(* IEC 61131-3 sources: SmartHomeNew/snapshots/2026-05-25 (part 2) *)

(* ---- GVL_SENSOR_CONSENSUS.gvl ---- *)
VAR_GLOBAL
    // Global sensor consensus authority.
    Sensor_Consensus_Valid : BOOL := FALSE;
    Sensor_Consensus_Quarantine_Active : BOOL := TRUE;
    Sensor_Consensus_Lease_Expired : BOOL := TRUE;

    // Physics-consistency proofs.
    Physics_Invariants_Satisfied : BOOL := FALSE;
    Cross_Sensor_Correlation_Valid : BOOL := FALSE;
    Telemetry_Plausibility_Valid : BOOL := FALSE;

    // Divergence detection.
    Sensor_Drift_Detected : BOOL := FALSE;
    Sensor_Partition_Detected : BOOL := FALSE;
    Sensor_Hallucination_Suspected : BOOL := FALSE;
    Cross_Sensor_Divergence_Detected : BOOL := FALSE;

    // Physical causality consistency.
    Flow_Response_Valid : BOOL := FALSE;
    Pressure_Response_Valid : BOOL := FALSE;
    Airflow_Response_Valid : BOOL := FALSE;
    Current_Signature_Valid : BOOL := FALSE;

    // Consensus temporal authority.
    Sensor_Consensus_Epoch : UDINT := 0;
    Last_Consensus_Update_MS : UDINT := 0;
    Sensor_Consensus_Freshness_Valid : BOOL := FALSE;

    // Oscillation/drift containment.
    Sensor_Oscillation_Detected : BOOL := FALSE;
    Sensor_Stuck_State_Detected : BOOL := FALSE;
    Sensor_Replay_Suspected : BOOL := FALSE;

    // Diagnostics.
    Sensor_Consensus_Last_Error_Code : UDINT := 0;
    Sensor_Consensus_Last_Error_Text : STRING(160) := '';
    Sensor_Consensus_Invalidation_Count : UDINT := 0;
END_VAR

(* ---- GVL_STATE.gvl ---- *)
{attribute 'qualified_only'}
VAR_GLOBAL
    G_Floor_Temps : ARRAY[1..GVL_CONSTANTS.C_MAX_HEATING_CIRCUITS] OF REAL;
    G_Room_Temps : ARRAY[1..GVL_CONSTANTS.C_MAX_ZONES] OF REAL;
    G_Last_Valid_Room_Temps : ARRAY[1..GVL_CONSTANTS.C_MAX_ZONES] OF REAL;
    G_Last_Valid_Floor_Temps : ARRAY[1..GVL_CONSTANTS.C_MAX_HEATING_CIRCUITS] OF REAL;
    G_Temp_Sensor_Fault : ARRAY[1..GVL_CONSTANTS.C_MAX_ZONES] OF BOOL;
    G_Floor_Temp_Sensor_Fault : ARRAY[1..GVL_CONSTANTS.C_MAX_HEATING_CIRCUITS] OF BOOL;
    G_Room_Hum : ARRAY[1..GVL_CONSTANTS.C_MAX_ZONES] OF REAL;
    G_Room_CO2 : ARRAY[1..GVL_CONSTANTS.C_MAX_ZONES] OF REAL;
    G_Motion_Sensors : ARRAY[1..GVL_CONSTANTS.C_MAX_LIGHT_ZONES] OF BOOL;
    G_Door_Sensors : ARRAY[1..GVL_CONSTANTS.C_MAX_DOOR_SENSORS] OF BOOL;
    G_Window_Sensors : ARRAY[1..GVL_CONSTANTS.C_MAX_ZONES] OF BOOL;
    G_Water_Sensors : ARRAY[1..GVL_CONSTANTS.C_MAX_FLOOD_SENSORS] OF BOOL;
    G_Flood_Warning : ARRAY[1..GVL_CONSTANTS.C_MAX_FLOOD_SENSORS] OF BOOL;
    G_Flood_Alarm : ARRAY[1..GVL_CONSTANTS.C_MAX_FLOOD_SENSORS] OF BOOL;
    G_Flood_Warning_Rise : ARRAY[1..GVL_CONSTANTS.C_MAX_FLOOD_SENSORS] OF BOOL;
    G_Flood_Alarm_Rise : ARRAY[1..GVL_CONSTANTS.C_MAX_FLOOD_SENSORS] OF BOOL;
    G_Flood_Alarm_Fall : ARRAY[1..GVL_CONSTANTS.C_MAX_FLOOD_SENSORS] OF BOOL;
    G_Smoke_Sensors : ARRAY[1..GVL_CONSTANTS.C_MAX_SMOKE_SENSORS] OF BOOL;
    G_Methane_Sensors : ARRAY[1..GVL_CONSTANTS.C_MAX_METHANE_SENSORS] OF REAL;
    G_CO_Sensors : ARRAY[1..GVL_CONSTANTS.C_MAX_CO_SENSORS] OF REAL;
    G_Manifold_Pressures : ARRAY[1..GVL_CONSTANTS.C_MAX_MANIFOLDS] OF REAL;
    G_Manifold_Currents : ARRAY[1..GVL_CONSTANTS.C_MAX_MANIFOLDS] OF REAL;
    G_Predictive_Pump_Pressure_Drop : ARRAY[1..GVL_CONSTANTS.C_MAX_MANIFOLDS] OF BOOL;
    G_Predictive_Pump_Current_Rise : ARRAY[1..GVL_CONSTANTS.C_MAX_MANIFOLDS] OF BOOL;
    G_Manifold_T_Supply : ARRAY[1..GVL_CONSTANTS.C_MAX_MANIFOLDS] OF REAL;
    G_Manifold_T_Return : ARRAY[1..GVL_CONSTANTS.C_MAX_MANIFOLDS] OF REAL;
    G_Boiler_Flame : ARRAY[1..GVL_CONSTANTS.C_MAX_BOILERS] OF BOOL;
    G_Boiler_Error : ARRAY[1..GVL_CONSTANTS.C_MAX_BOILERS] OF BOOL;
    G_Boiler_OT_Online : ARRAY[1..GVL_CONSTANTS.C_MAX_BOILERS] OF BOOL;
    G_Boiler_OT_Command_Ack : ARRAY[1..GVL_CONSTANTS.C_MAX_BOILERS] OF BOOL;
    G_Boiler_OT_Command_Timeout : ARRAY[1..GVL_CONSTANTS.C_MAX_BOILERS] OF BOOL;
    G_Boiler_OT_Heartbeat_Timeout : ARRAY[1..GVL_CONSTANTS.C_MAX_BOILERS] OF BOOL;
    G_Boiler_OT_Adapter_Error : ARRAY[1..GVL_CONSTANTS.C_MAX_BOILERS] OF BOOL;
    G_Boiler_OT_Heartbeat_Age_MS : ARRAY[1..GVL_CONSTANTS.C_MAX_BOILERS] OF UDINT;
    G_Boiler_OT_Command_Age_MS : ARRAY[1..GVL_CONSTANTS.C_MAX_BOILERS] OF UDINT;
    G_Boiler_OT_Adapter_State : ARRAY[1..GVL_CONSTANTS.C_MAX_BOILERS] OF E_OpenTherm_Adapter_State;
    G_Boiler_OT_Error_State : ARRAY[1..GVL_CONSTANTS.C_MAX_BOILERS] OF E_OpenTherm_Error;
    G_Boiler_OT_Enable : ARRAY[1..GVL_CONSTANTS.C_MAX_BOILERS] OF BOOL;
    G_Boiler_OT_Setpoint : ARRAY[1..GVL_CONSTANTS.C_MAX_BOILERS] OF REAL;
    G_Heating_Cascade_Available : BOOL;
    G_Heating_Cascade_Degraded : BOOL;
    G_Heating_Cascade_Partial_Capacity : BOOL;
    G_Heating_Cascade_No_Flame : BOOL;
    G_Heating_Cascade_Transport_Degraded : BOOL;
    G_Heating_Cascade_Ignition_Timeout : BOOL;
    G_Heating_Cascade_Active_Boilers : UINT;
    G_Heating_Cascade_Available_Boilers : UINT;
    G_Physical_Switches : ARRAY[1..GVL_CONSTANTS.C_MAX_LIGHT_ZONES] OF BOOL;
    G_Socket_Switches : ARRAY[1..GVL_CONSTANTS.C_MAX_SOCKETS] OF BOOL;
    G_Outdoor_Temp : REAL;
    G_Ambient_Lux : REAL;
    G_Ambient_Lux_Valid : BOOL := FALSE;
    G_Ambient_Lux_Sensor_Fault : BOOL := FALSE;
    G_Supply_Temps : ARRAY[1..GVL_CONSTANTS.C_MAX_SUPPLY_TEMPS] OF REAL;
    G_DHW_Temp : REAL;
    G_DHW_Pressure : REAL;
    G_Zone_Valves : ARRAY[1..GVL_CONSTANTS.C_MAX_HEATING_CIRCUITS] OF BOOL;
    G_Manifold_Pumps : ARRAY[1..GVL_CONSTANTS.C_MAX_MANIFOLDS] OF BOOL;
    G_Manifold_Valves : ARRAY[1..GVL_CONSTANTS.C_MAX_MANIFOLDS] OF REAL;
    G_Manifold_End_Switches : ARRAY[1..GVL_CONSTANTS.C_MAX_MANIFOLDS] OF BOOL;
    G_Supply_Fans : ARRAY[1..GVL_CONSTANTS.C_MAX_SUPPLY_FANS] OF REAL;
    G_Exhaust_Fans : ARRAY[1..GVL_CONSTANTS.C_MAX_EXHAUST_FANS] OF REAL;
    G_Vent_Heater_Power : ARRAY[1..GVL_CONSTANTS.C_MAX_BOILERS] OF REAL;
    G_Lighting_Levels : ARRAY[1..GVL_CONSTANTS.C_MAX_LIGHT_ZONES] OF BYTE;
    G_Blinds_Positions : ARRAY[1..GVL_CONSTANTS.C_MAX_BLINDS] OF BYTE;
    G_Socket_States : ARRAY[1..GVL_CONSTANTS.C_MAX_SOCKETS] OF BOOL;
    G_DHW_Heating_Pump : BOOL;
    G_DHW_Circ_Pump : BOOL;
    G_Backup_Circulation_Pump : BOOL;
    G_Electric_Heater_Enable : BOOL;
    G_Safety_Gas_Alarm : BOOL;
    G_Safety_Leak_Alarm : BOOL;
    G_Safety_Smoke_Alarm : BOOL;
    G_Safety_Emergency_Stop : BOOL;
    G_Safety_Gas_Latched : BOOL;
    G_Safety_Leak_Latched : BOOL;
    G_Safety_Smoke_Latched : BOOL;
    G_Safety_Freeze_Risk : BOOL;
    G_System_Mode : E_System_Operating_Mode := E_System_Operating_Mode.MODE_NORMAL;
    G_System_Mode_Text : STRING(64);
    G_Heating_IO_Fault : BOOL;
    G_Heating_Sensor_Fault : BOOL;
    G_Heating_Subsystem_Degraded : BOOL;
    G_Allocation_Policy_Active : BOOL;
    G_Allocation_Freeze_Bypass_Active : BOOL;
    G_Allocation_DHW_Bypass_Active : BOOL;
    G_Allocation_Budget_Max : REAL;
    G_Allocation_Budget_Used : REAL;
    G_Allocation_Requested : ARRAY[1..GVL_CONSTANTS.C_MAX_MANIFOLDS] OF BOOL;
    G_Allocation_Allowed : ARRAY[1..GVL_CONSTANTS.C_MAX_MANIFOLDS] OF BOOL;
    G_Allocation_Filtered : ARRAY[1..GVL_CONSTANTS.C_MAX_MANIFOLDS] OF BOOL;
    G_Allocation_Block_Reason : ARRAY[1..GVL_CONSTANTS.C_MAX_MANIFOLDS] OF E_Heating_Allocation_Block_Reason;
    G_Allocation_Effective_Priority : ARRAY[1..GVL_CONSTANTS.C_MAX_MANIFOLDS] OF INT;
    G_Policy_Target_Adjustment_Active : BOOL;
    G_Policy_Target_Adjustment_Applied : REAL;
    G_Policy_Priority_Multiplier_Applied : REAL;
    G_Policy_Priority_Bridge_Active : BOOL;
    G_Policy_Priority_Bias_Applied : ARRAY[1..GVL_CONSTANTS.C_MAX_MANIFOLDS] OF REAL;
    G_Policy_Priority_Effective : ARRAY[1..GVL_CONSTANTS.C_MAX_MANIFOLDS] OF INT;
    G_Heating_RootCause : E_Heating_RootCause := E_Heating_RootCause.RC_NONE;
    G_Heating_RootConfidence : REAL;
    G_Heating_Confidence : REAL := 1.0;
    G_Heating_Error_Score : REAL := 0.0;
    G_Heating_Confidence_Reason_Code : INT := 0;
    G_Heating_Confidence_Reason_Text : STRING(128) := 'OK';
    G_DHW_IO_Fault : BOOL;
    G_DHW_Sensor_Fault : BOOL;
    G_DHW_Subsystem_Degraded : BOOL;
    G_Ventilation_IO_Fault : BOOL;
    G_Ventilation_Subsystem_Degraded : BOOL;
    G_Lighting_IO_Fault : BOOL;
    G_Lighting_Subsystem_Degraded : BOOL;
    G_Access_Comm_Fault : BOOL;
    G_Evacuation_Lighting_Active : BOOL;
    G_Evac_Hazard_Zone : ARRAY[1..GVL_CONSTANTS.C_MAX_LIGHT_ZONES] OF BOOL;
    G_Evac_Guidance : ARRAY[1..GVL_CONSTANTS.C_MAX_LIGHT_ZONES] OF INT;
    G_Rule_Actions : ARRAY[1..GVL_CONSTANTS.C_MAX_RULES] OF ST_Rule_Action;
    G_Sim_Lights : ARRAY[1..GVL_CONSTANTS.C_MAX_LIGHT_ZONES] OF BOOL;
    G_Freeze_Hardware_Degraded : BOOL;
    G_Freeze_Hardware_Failed : BOOL;
    G_Water_Zone_Enable : ARRAY[1..GVL_CONSTANTS.C_MAX_WATER_ZONES] OF BOOL;
    G_Water_Zone_Open_FB : ARRAY[1..GVL_CONSTANTS.C_MAX_WATER_ZONES] OF BOOL;
    G_Water_Zone_Close_FB : ARRAY[1..GVL_CONSTANTS.C_MAX_WATER_ZONES] OF BOOL;
    G_Water_Zone_Exercise_Active : ARRAY[1..GVL_CONSTANTS.C_MAX_WATER_ZONES] OF BOOL;
    G_Preheat_Request : BOOL;
    G_Freeze_Request : BOOL;
    G_Target_Temperature : REAL;
END_VAR

(* ---- GVL_SYSTEM_HEALTH.gvl ---- *)
VAR_GLOBAL
    G_First_Fault_Active : BOOL;
    G_First_Fault_Type : INT;
    G_First_Fault_Source : INT;
    G_System_Severity : E_System_Severity;
    G_Root_Cause : E_System_Root_Cause;
    G_Watchdog_Fault : BOOL;
END_VAR

(* ---- GVL_TIME_SERVICE.gvl ---- *)
{attribute 'qualified_only'}
VAR_GLOBAL
    // Published effective time for consumers
    G_Now_MS : UDINT;
    G_Time_Of_Day_MS : UDINT;
    G_Current_TOD : TOD;
    G_Day_Of_Week : INT;
    G_Last_Now_MS : UDINT;
    G_Delta_MS : UDINT;
    G_Wrap_Detected : BOOL;

    // Simulation controls (HMI/runtime configurable)
    G_Sim_Enabled : BOOL;
    G_Sim_Frozen : BOOL;
    G_Sim_Time_Scale : REAL := 1.0;
    G_Sim_Now_MS : UDINT;
    G_Sim_Time_Of_Day_MS : UDINT;
    G_Sim_Day_Of_Week : INT := 1;
END_VAR

(* ---- GVL_TRUST_EPOCH_MONOTONICITY_FABRIC.gvl ---- *)
VAR_GLOBAL
    // Deterministic trust epoch monotonicity governance.
    Trust_Epoch_Monotonicity_Valid : BOOL := FALSE;
    Trust_Epoch_Monotonicity_Granted : BOOL := FALSE;
    Trust_Epoch_Monotonicity_Quarantine_Active : BOOL := TRUE;

    // Monotonic trust continuity proofs.
    Global_Trust_Epoch_Monotonic : BOOL := FALSE;
    Rollback_Resistant_Authority_Valid : BOOL := FALSE;
    Recovery_Epoch_Strictly_Newer : BOOL := FALSE;
    Distributed_Trust_Vector_Coherent : BOOL := FALSE;
    Irreversible_Trust_Progression_Stable : BOOL := FALSE;

    // Distributed temporal trust integrity.
    CrossNode_Trust_Epoch_Aligned : BOOL := FALSE;
    Recovery_Timeline_Dominance_Valid : BOOL := FALSE;
    Federation_Epoch_Progression_Coherent : BOOL := FALSE;
    Trust_Revocation_History_Monotonic : BOOL := FALSE;

    // Temporal trust rollback detectors.
    Temporal_Trust_Rollback_Detected : BOOL := FALSE;
    Replay_Authority_Epoch_Detected : BOOL := FALSE;
    CrossNode_Trust_Vector_Regression : BOOL := FALSE;
    Stale_Federation_Epoch_Rejoin : BOOL := FALSE;
    Recovery_Timeline_Fork_Detected : BOOL := FALSE;
    Revoked_Epoch_Resurrection_Detected : BOOL := FALSE;

    // Monotonicity epochs.
    Trust_Epoch_Monotonicity_Epoch : UDINT := 0;
    Trust_Epoch_Monotonicity_Epoch_Coherent : BOOL := FALSE;

    // Temporal authority.
    Trust_Epoch_Monotonicity_Last_Update_MS : UDINT := 0;
    Trust_Epoch_Monotonicity_Lease_Expired : BOOL := TRUE;

    // Diagnostics.
    Trust_Epoch_Monotonicity_Last_Error_Code : UDINT := 0;
    Trust_Epoch_Monotonicity_Last_Error_Text : STRING(160) := '';
    Trust_Epoch_Monotonicity_Invalidation_Count : UDINT := 0;
END_VAR

(* ---- GVL_WATER_DOMAIN_STATUS.gvl ---- *)
{attribute 'qualified_only'}
VAR_GLOBAL
    // Water domain status. Observational only.

    G_Runtime_Required : BOOL := FALSE;
    G_Runtime_Executed : BOOL := FALSE;
    G_Runtime_Idle_By_Design : BOOL := FALSE;
    G_Recovery_Requested : BOOL := FALSE;
    G_Global_Path_Active : BOOL := FALSE;
    G_Output_35_Active : BOOL := FALSE;
    G_Output_36_Active : BOOL := FALSE;
    G_Any_Zone_Active : BOOL := FALSE;
    G_Last_Update_MS : UDINT := 0;
    G_Status_Code : UINT := 0;
    G_Status_Text : STRING(128) := '';
END_VAR

(* ---- GVL_Water_Isolation_Intent.gvl ---- *)
{attribute 'qualified_only'}
VAR_GLOBAL
    // ==============================================================================
    // Water/Flood isolation intent publication.
    // ==============================================================================
    //
    // Explicit authority augmentation layer.
    //
    // This layer publishes:
    // - selective isolation intent;
    // - per-zone close requests;
    // - fallback-to-global requirements.
    //
    // It does NOT directly own outputs.
    // Final authority remains inside runtime arbitration/safety layers.
    // ==============================================================================

    // Per-zone isolation intent.
    G_Zone_Close_Requested : ARRAY[1..GVL_CONSTANTS.C_MAX_FLOOD_SENSORS] OF BOOL;

    // Valve-group visibility.
    G_Valve_Group_Close_Requested : ARRAY[1..GVL_CONSTANTS.C_MAX_FLOOD_SENSORS] OF BOOL;

    // Conservative fallback visibility.
    G_Global_Isolation_Requested : BOOL;

    // Explainability.
    G_Intent_Valid : BOOL;
    G_Status_Code : UINT;
    G_Status_Text : STRING(128);
END_VAR

(* ---- GVL_WATER_OUTPUT.gvl ---- *)
VAR_GLOBAL
    // Global inlet valves.
    // 35 = общий ввод ХВС, 36 = общий ввод ГВС.
    DO_Water_Valve_35_Open : BOOL := FALSE;
    DO_Water_Valve_35_Close : BOOL := FALSE;
    DO_Water_Valve_36_Open : BOOL := FALSE;
    DO_Water_Valve_36_Close : BOOL := FALSE;

    // Local riser motorized ball valves with end switches.
    // 1 = стояк 1 ХВС, 2 = стояк 1 ГВС,
    // 3 = стояк 2 ХВС, 4 = стояк 2 ГВС,
    // 5 = стояк 3 ХВС, 6 = стояк 3 ГВС.
    DO_Water_Local_Valve_Open : ARRAY[1..6] OF BOOL;
    DO_Water_Local_Valve_Close : ARRAY[1..6] OF BOOL;

    DO_Water_Zone_Enable : ARRAY[1..GVL_CONSTANTS.C_MAX_WATER_ZONES] OF BOOL;
END_VAR

(* ---- GVL_Water_Topology_Config.gvl ---- *)
{attribute 'qualified_only'}
VAR_GLOBAL
    G_Config_Record : ARRAY[1..64] OF ST_Water_Topology_Config_Record;

    G_Active_Config_Version : UDINT;
    G_Config_Loaded : BOOL;
    G_Runtime_Remap_Ready : BOOL;

    G_Any_Invalid_Config : BOOL;
    G_Any_Multi_Valve_Required : BOOL;

    G_Runtime_Valid : BOOL;
    G_Last_Update_MS : UDINT;

    G_Status_Code : UINT;
    G_Status_Text : STRING(128);
END_VAR

(* ---- GVL_Water_Valve_Runtime.gvl ---- *)
{attribute 'qualified_only'}
VAR_GLOBAL
    // ==============================================================================
    // Water/Flood valve governance publication.
    // ==============================================================================
    //
    // Observe-first valve governance and confirmation visibility.
    //
    // This layer publishes:
    // - valve runtime semantics;
    // - authority visibility;
    // - confirmation semantics;
    // - degraded-state visibility.
    //
    // This layer does NOT directly own physical outputs.
    // ==============================================================================

    G_Valve_Runtime_State : ARRAY[1..64] OF ST_Water_Valve_Runtime_State;

    // Aggregated visibility.
    G_Any_Valve_Degraded : BOOL;
    G_Any_Confirmation_Unknown : BOOL;
    G_Any_Unsafe_Reopen_Denied : BOOL;

    // Lifecycle.
    G_Runtime_Valid : BOOL;
    G_Last_Update_MS : UDINT;

    // Explainability.
    G_Status_Code : UINT;
    G_Status_Text : STRING(128);
END_VAR

(* ---- FB_Access_Pulse_Channel.st ---- *)
FUNCTION_BLOCK FB_Access_Pulse_Channel
VAR_INPUT
    VI_Command : BOOL;
    VI_Reset : BOOL;
    VI_Now_MS : UDINT;
    VI_Pulse_MS : UDINT;
END_VAR
VAR_OUTPUT
    VO_Output : BOOL;
    VO_Active : BOOL;
END_VAR
VAR
    L_Prev_Command : BOOL;
    L_Start_MS : UDINT;
    L_Elapsed_MS : UDINT;
END_VAR

IF VI_Reset THEN
    VO_Output := FALSE;
    VO_Active := FALSE;
    L_Prev_Command := VI_Command;
    L_Start_MS := VI_Now_MS;
    RETURN;
END_IF;

IF VI_Command AND NOT L_Prev_Command THEN
    VO_Active := TRUE;
    L_Start_MS := VI_Now_MS;
END_IF;

VO_Output := FALSE;

IF VO_Active THEN
    IF VI_Now_MS >= L_Start_MS THEN
        L_Elapsed_MS := VI_Now_MS - L_Start_MS;
    ELSE
        L_Elapsed_MS := (4294967295 - L_Start_MS) + VI_Now_MS + 1;
    END_IF;

    IF L_Elapsed_MS < VI_Pulse_MS THEN
        VO_Output := TRUE;
    ELSE
        VO_Active := FALSE;
    END_IF;
END_IF;

L_Prev_Command := VI_Command;

END_FUNCTION_BLOCK
// >>> BULK_SYNC_ANCHOR: FB_Access_Pulse_Channel <<<

(* ---- FB_Alarm_Manager.st ---- *)
FUNCTION_BLOCK FB_Alarm_Manager
VAR_INPUT
    VI_System_Time_MS : UDINT; // Системное время (мс)
    VI_IsActivePLC : BOOL; // Флаг: Данный ПЛК является ведущим

    // Входы от подсистем
    VI_Gas_Alarm : BOOL; // Сигнал тревоги: Утечка газа
    VI_Fire_Alarm : BOOL; // Сигнал тревоги: Пожар
    VI_Flood_Alarm : BOOL; // Сигнал тревоги: Протечка воды
    VI_Security_Alarm : BOOL; // Сигнал тревоги: Охранная система
    VI_First_Fault_Active : BOOL; // Активна защёлкнутая первая причина деградации
    VI_First_Fault_Type : INT; // 1=IO,2=Sensor,3=Comm,4=Subsystem
    VI_First_Fault_Source : INT; // 1=Heating,2=DHW,3=Ventilation,4=Lighting,5=Access

    // Сообщения от подсистем (для детализации)
    VI_Security_Msg : STRING(200); // Детальное сообщение от охранной системы

    // Команды с HMI
    VI_Acknowledge_All : BOOL; // Команда: Квитировать все тревоги
    VI_Mute_Siren : BOOL; // Команда: Временное отключение сирены
END_VAR
VAR_IN_OUT
    VI_Boiler_Errors : ARRAY[1..GVL_CONSTANTS.C_MAX_BOILERS] OF BOOL; // Ошибки котлов
END_VAR
VAR_IN_OUT
    VIO_Next_Alarm_ID : UDINT; // Глобальный счетчик ID тревог
END_VAR
VAR_OUTPUT
    VO_Global_Critical : BOOL; // Есть неквитированные критические аварии
    VO_Global_Warning : BOOL;  // Есть неквитированные предупреждения
    VO_Siren_Active : BOOL;    // Требуется включение сирены
    VO_Active_Count : INT;     // Количество активных тревог
    VO_Unacked_Count : INT;    // Количество неквитированных тревог
    VO_Event_Pulse : BOOL;     // Пульс события для History bridge
    VO_Event_Code : UDINT;     // 1201=ack all, 1202=alarm cleared, 1203=alarm created
    VO_Event_Value : REAL;     // Доп. значение события

    VO_Alarm_List : ARRAY[1..GVL_CONSTANTS.C_MAX_ALARMS] OF ST_Alarm_Record; // Список активных тревог для HMI
END_VAR
VAR
    L_i, L_j, L_k : INT;
    L_Target_Slot : INT;
    L_Min_Pri : INT;
    L_Pending_Alarms : ARRAY[1..10] OF ST_Alarm_Record;
    L_Pending_Count : INT := 0;

    // Фронты и антидребезг для детекции новых тревог
    T_Debounce_Gas : FB_System_Timer;
    T_Debounce_Fire : FB_System_Timer;
    T_Debounce_Flood : FB_System_Timer;
    T_Debounce_Security : FB_System_Timer;
    R_Trig_Gas : R_TRIG;
    R_Trig_Fire : R_TRIG;
    R_Trig_Flood : R_TRIG;
    R_Trig_Security : R_TRIG;
    R_Trig_First_Fault : R_TRIG;
    R_Trig_Boiler : ARRAY[1..GVL_CONSTANTS.C_MAX_BOILERS] OF R_TRIG;
    L_First_Fault_Source_Text : STRING(32);
    L_First_Fault_Type_Text : STRING(32);
    L_Event_Pulse_Latched : BOOL;
END_VAR

VO_Event_Pulse := FALSE;
VO_Event_Code := 0;
VO_Event_Value := 0.0;

// 1. Детекция новых тревог (антидребезг + передний фронт)
T_Debounce_Gas(IN := VI_Gas_Alarm, PT := T#100ms, VI_System_Time_MS := VI_System_Time_MS);
T_Debounce_Fire(IN := VI_Fire_Alarm, PT := T#100ms, VI_System_Time_MS := VI_System_Time_MS);
T_Debounce_Flood(IN := VI_Flood_Alarm, PT := T#500ms, VI_System_Time_MS := VI_System_Time_MS);
T_Debounce_Security(IN := VI_Security_Alarm, PT := T#100ms, VI_System_Time_MS := VI_System_Time_MS);

R_Trig_Gas(CLK := T_Debounce_Gas.Q);
R_Trig_Fire(CLK := T_Debounce_Fire.Q);
R_Trig_Flood(CLK := T_Debounce_Flood.Q);
R_Trig_Security(CLK := T_Debounce_Security.Q);
R_Trig_First_Fault(CLK := VI_First_Fault_Active);
FOR L_i := 1 TO GVL_CONSTANTS.C_MAX_BOILERS DO
    R_Trig_Boiler[L_i](CLK := VI_Boiler_Errors[L_i]);
END_FOR;

// 2. Добавление новых тревог в список (Кольцевой буфер)
L_Pending_Count := 0;
L_Event_Pulse_Latched := FALSE;

IF R_Trig_Gas.Q AND L_Pending_Count < 10 THEN
    L_Pending_Count := L_Pending_Count + 1;
    L_Pending_Alarms[L_Pending_Count].Timestamp_MS := VI_System_Time_MS;
    L_Pending_Alarms[L_Pending_Count].Source := 'Gas';
    L_Pending_Alarms[L_Pending_Count].Source_ID := 0;
    L_Pending_Alarms[L_Pending_Count].Message := 'Критическая концентрация газа!';
    L_Pending_Alarms[L_Pending_Count].Severity := E_ALERT_PRIORITY.ALERT_PRIORITY_CRITICAL;
    L_Pending_Alarms[L_Pending_Count].Is_Active := TRUE;
    L_Pending_Alarms[L_Pending_Count].Is_Acknowledged := FALSE;
END_IF;

IF R_Trig_Fire.Q AND L_Pending_Count < 10 THEN
    L_Pending_Count := L_Pending_Count + 1;
    L_Pending_Alarms[L_Pending_Count].Timestamp_MS := VI_System_Time_MS;
    L_Pending_Alarms[L_Pending_Count].Source := 'Fire';
    L_Pending_Alarms[L_Pending_Count].Source_ID := 0;
    L_Pending_Alarms[L_Pending_Count].Message := 'Обнаружено задымление!';
    L_Pending_Alarms[L_Pending_Count].Severity := E_ALERT_PRIORITY.ALERT_PRIORITY_CRITICAL;
    L_Pending_Alarms[L_Pending_Count].Is_Active := TRUE;
    L_Pending_Alarms[L_Pending_Count].Is_Acknowledged := FALSE;
END_IF;

IF R_Trig_Flood.Q AND L_Pending_Count < 10 THEN
    L_Pending_Count := L_Pending_Count + 1;
    L_Pending_Alarms[L_Pending_Count].Timestamp_MS := VI_System_Time_MS;
    L_Pending_Alarms[L_Pending_Count].Source := 'Flood';
    L_Pending_Alarms[L_Pending_Count].Source_ID := 0;
    L_Pending_Alarms[L_Pending_Count].Message := 'Обнаружена протечка воды!';
    L_Pending_Alarms[L_Pending_Count].Severity := E_ALERT_PRIORITY.ALERT_PRIORITY_CRITICAL;
    L_Pending_Alarms[L_Pending_Count].Is_Active := TRUE;
    L_Pending_Alarms[L_Pending_Count].Is_Acknowledged := FALSE;
END_IF;

IF R_Trig_Security.Q AND L_Pending_Count < 10 THEN
    L_Pending_Count := L_Pending_Count + 1;
    L_Pending_Alarms[L_Pending_Count].Timestamp_MS := VI_System_Time_MS;
    L_Pending_Alarms[L_Pending_Count].Source := 'Security';
    L_Pending_Alarms[L_Pending_Count].Source_ID := 0;
    L_Pending_Alarms[L_Pending_Count].Message := VI_Security_Msg;
    L_Pending_Alarms[L_Pending_Count].Severity := E_ALERT_PRIORITY.ALERT_PRIORITY_CRITICAL;
    L_Pending_Alarms[L_Pending_Count].Is_Active := TRUE;
    L_Pending_Alarms[L_Pending_Count].Is_Acknowledged := FALSE;
END_IF;

IF R_Trig_First_Fault.Q AND L_Pending_Count < 10 THEN
    L_Pending_Count := L_Pending_Count + 1;
    L_Pending_Alarms[L_Pending_Count].Timestamp_MS := VI_System_Time_MS;
    L_Pending_Alarms[L_Pending_Count].Source := 'Diagnostics';
    L_Pending_Alarms[L_Pending_Count].Source_ID := TO_BYTE(VI_First_Fault_Source);

    CASE VI_First_Fault_Type OF
        1: L_First_Fault_Type_Text := 'IO';
        2: L_First_Fault_Type_Text := 'Sensor';
        3: L_First_Fault_Type_Text := 'Comm';
        4: L_First_Fault_Type_Text := 'Subsystem';
        ELSE L_First_Fault_Type_Text := 'Unknown';
    END_CASE;

    CASE VI_First_Fault_Source OF
        1: L_First_Fault_Source_Text := 'Heating';
        2: L_First_Fault_Source_Text := 'DHW';
        3: L_First_Fault_Source_Text := 'Ventilation';
        4: L_First_Fault_Source_Text := 'Lighting';
        5: L_First_Fault_Source_Text := 'Access';
        ELSE L_First_Fault_Source_Text := 'Unknown';
    END_CASE;

    L_Pending_Alarms[L_Pending_Count].Message := CONCAT('Diagnostics root cause: ', CONCAT(L_First_Fault_Source_Text, CONCAT(' / ', L_First_Fault_Type_Text)));
    L_Pending_Alarms[L_Pending_Count].Severity := E_ALERT_PRIORITY.ALERT_PRIORITY_HIGH;
    L_Pending_Alarms[L_Pending_Count].Is_Active := TRUE;
    L_Pending_Alarms[L_Pending_Count].Is_Acknowledged := FALSE;
END_IF;

FOR L_j := 1 TO GVL_CONSTANTS.C_MAX_BOILERS DO
    IF R_Trig_Boiler[L_j].Q AND L_Pending_Count < 10 THEN
        L_Pending_Count := L_Pending_Count + 1;
        L_Pending_Alarms[L_Pending_Count].Timestamp_MS := VI_System_Time_MS;
        L_Pending_Alarms[L_Pending_Count].Source := 'Boiler';
        L_Pending_Alarms[L_Pending_Count].Source_ID := TO_BYTE(L_j);
        L_Pending_Alarms[L_Pending_Count].Message := CONCAT('Авария котла №', INT_TO_STRING(L_j));
        L_Pending_Alarms[L_Pending_Count].Severity := E_ALERT_PRIORITY.ALERT_PRIORITY_HIGH;
        L_Pending_Alarms[L_Pending_Count].Is_Active := TRUE;
        L_Pending_Alarms[L_Pending_Count].Is_Acknowledged := FALSE;
    END_IF;
END_FOR;

// Обработка очереди новых тревог с учетом приоритетов
FOR L_i := 1 TO L_Pending_Count DO

    L_Target_Slot := 0;

    // 1. Ищем пустой слот
    FOR L_k := 1 TO GVL_CONSTANTS.C_MAX_ALARMS DO
        IF VO_Alarm_List[L_k].ID = 0 THEN
            L_Target_Slot := L_k;
            EXIT;
        END_IF;
    END_FOR;

    // 2. Ищем квитированную тревогу с наименьшим приоритетом
    IF L_Target_Slot = 0 THEN
        L_Min_Pri := 999;
        FOR L_k := 1 TO GVL_CONSTANTS.C_MAX_ALARMS DO
            IF VO_Alarm_List[L_k].Is_Acknowledged AND TO_INT(VO_Alarm_List[L_k].Severity) < L_Min_Pri THEN
                L_Min_Pri := TO_INT(VO_Alarm_List[L_k].Severity);
                L_Target_Slot := L_k;
            END_IF;
        END_FOR;
    END_IF;

    // 3. Ищем неквитированную тревогу с наименьшим приоритетом (если он ниже добавляемой)
    IF L_Target_Slot = 0 THEN
        L_Min_Pri := 999;
        FOR L_k := 1 TO GVL_CONSTANTS.C_MAX_ALARMS DO
            IF TO_INT(VO_Alarm_List[L_k].Severity) < L_Min_Pri AND TO_INT(VO_Alarm_List[L_k].Severity) < TO_INT(L_Pending_Alarms[L_i].Severity) THEN
                L_Min_Pri := TO_INT(VO_Alarm_List[L_k].Severity);
                L_Target_Slot := L_k;
            END_IF;
        END_FOR;
    END_IF;

    IF L_Target_Slot = 0 THEN
        // Буфер полон критических неквитированных тревог. Не затираем!
        CONTINUE;
    END_IF;

    VO_Alarm_List[L_Target_Slot] := L_Pending_Alarms[L_i];
    VO_Alarm_List[L_Target_Slot].ID := VIO_Next_Alarm_ID;
    VIO_Next_Alarm_ID := VIO_Next_Alarm_ID + 1;
    IF VIO_Next_Alarm_ID = 0 THEN VIO_Next_Alarm_ID := 1; END_IF;
    IF NOT L_Event_Pulse_Latched THEN
        VO_Event_Pulse := TRUE;
        VO_Event_Code := 1203;
        VO_Event_Value := TO_REAL(VO_Alarm_List[L_Target_Slot].Severity);
        L_Event_Pulse_Latched := TRUE;
    END_IF;
END_FOR;

// 3. Обновление статуса существующих тревог (ушли ли они?)
FOR L_i := 1 TO GVL_CONSTANTS.C_MAX_ALARMS DO
    IF VO_Alarm_List[L_i].ID <> 0 THEN
        IF VO_Alarm_List[L_i].Source = 'Gas' THEN VO_Alarm_List[L_i].Is_Active := VI_Gas_Alarm;
        ELSIF VO_Alarm_List[L_i].Source = 'Fire' THEN VO_Alarm_List[L_i].Is_Active := VI_Fire_Alarm;
        ELSIF VO_Alarm_List[L_i].Source = 'Flood' THEN VO_Alarm_List[L_i].Is_Active := VI_Flood_Alarm;
        ELSIF VO_Alarm_List[L_i].Source = 'Security' THEN VO_Alarm_List[L_i].Is_Active := VI_Security_Alarm;
        ELSIF VO_Alarm_List[L_i].Source = 'Diagnostics' THEN VO_Alarm_List[L_i].Is_Active := VI_First_Fault_Active;
        ELSIF VO_Alarm_List[L_i].Source = 'Boiler' THEN
            IF TO_INT(VO_Alarm_List[L_i].Source_ID) >= 1 AND TO_INT(VO_Alarm_List[L_i].Source_ID) <= GVL_CONSTANTS.C_MAX_BOILERS THEN
                VO_Alarm_List[L_i].Is_Active := VI_Boiler_Errors[TO_INT(VO_Alarm_List[L_i].Source_ID)];
            END_IF;
        END_IF;
    END_IF;
END_FOR;

// 4. Квитирование тревог
IF VI_Acknowledge_All THEN
    FOR L_i := 1 TO GVL_CONSTANTS.C_MAX_ALARMS DO
        IF VO_Alarm_List[L_i].ID <> 0 THEN
            VO_Alarm_List[L_i].Is_Acknowledged := TRUE;
        END_IF;
    END_FOR;

    IF NOT L_Event_Pulse_Latched THEN
        VO_Event_Pulse := TRUE;
        VO_Event_Code := 1201;
        VO_Event_Value := TO_REAL(VO_Unacked_Count);
        L_Event_Pulse_Latched := TRUE;
    END_IF;
END_IF;

// 4.5 Автоквитирование некритичных тревог, если они больше не активны
FOR L_i := 1 TO GVL_CONSTANTS.C_MAX_ALARMS DO
    IF VO_Alarm_List[L_i].ID <> 0 AND NOT VO_Alarm_List[L_i].Is_Active AND NOT VO_Alarm_List[L_i].Is_Acknowledged THEN
        IF VO_Alarm_List[L_i].Severity <> E_ALERT_PRIORITY.ALERT_PRIORITY_CRITICAL THEN
            VO_Alarm_List[L_i].Is_Acknowledged := TRUE;
        END_IF;
    END_IF;
END_FOR;

// 5. Очистка списка (удаление неактивных И квитированных тревог)
// В кольцевом буфере мы просто помечаем слот как пустой (ID = 0), без сдвига массива
FOR L_i := 1 TO GVL_CONSTANTS.C_MAX_ALARMS DO
    IF VO_Alarm_List[L_i].ID <> 0 AND NOT VO_Alarm_List[L_i].Is_Active AND VO_Alarm_List[L_i].Is_Acknowledged THEN
        // Удаляем тревогу
        VO_Alarm_List[L_i].ID := 0;
        IF NOT L_Event_Pulse_Latched THEN
            VO_Event_Pulse := TRUE;
            VO_Event_Code := 1202;
            VO_Event_Value := 0.0;
            L_Event_Pulse_Latched := TRUE;
        END_IF;
    END_IF;
END_FOR;

// 6. Подсчет статистики и формирование глобальных флагов
VO_Global_Critical := FALSE;
VO_Global_Warning := FALSE;
VO_Siren_Active := FALSE;
VO_Active_Count := 0;
VO_Unacked_Count := 0;

FOR L_i := 1 TO GVL_CONSTANTS.C_MAX_ALARMS DO
    IF VO_Alarm_List[L_i].ID <> 0 THEN
        IF VO_Alarm_List[L_i].Is_Active THEN
            VO_Active_Count := VO_Active_Count + 1;
        END_IF;

        IF NOT VO_Alarm_List[L_i].Is_Acknowledged THEN
            VO_Unacked_Count := VO_Unacked_Count + 1;

            IF VO_Alarm_List[L_i].Severity = E_ALERT_PRIORITY.ALERT_PRIORITY_CRITICAL THEN
                VO_Global_Critical := TRUE;
                // Сирена работает только для активных неквитированных критических тревог, если не включен Mute
                IF VO_Alarm_List[L_i].Is_Active AND NOT VI_Mute_Siren THEN
                    VO_Siren_Active := TRUE;
                END_IF;
            ELSIF VO_Alarm_List[L_i].Severity = E_ALERT_PRIORITY.ALERT_PRIORITY_HIGH THEN
                VO_Global_Warning := TRUE;
            END_IF;
        END_IF;
    END_IF;
END_FOR;
// >>> BULK_SYNC_ANCHOR: FB_Alarm_Manager <<<
END_FUNCTION_BLOCK

(* ---- FB_Analog_Validator.st ---- *)
FUNCTION_BLOCK FB_Analog_Validator
VAR_INPUT
    VI_Value : REAL;
    VI_Min_Valid : REAL;
    VI_Max_Valid : REAL;
    VI_Fallback_Mode : INT := 0; // 0: Hold last good, 1: Default value
    VI_Default_Value : REAL := 0.0;
END_VAR
VAR_OUTPUT
    VO_Value : REAL;
    VO_Error : BOOL;
END_VAR
VAR
    L_Last_Good_Value : REAL;
    L_First_Valid : BOOL := FALSE;
END_VAR

IF VI_Value >= VI_Min_Valid AND VI_Value <= VI_Max_Valid THEN
    VO_Error := FALSE;
    VO_Value := VI_Value;
    L_Last_Good_Value := VI_Value;
    L_First_Valid := TRUE;
ELSE
    VO_Error := TRUE;
    IF VI_Fallback_Mode = 1 OR NOT L_First_Valid THEN
        VO_Value := VI_Default_Value;
    ELSE
        VO_Value := L_Last_Good_Value;
    END_IF;
END_IF;
// >>> BULK_SYNC_ANCHOR: FB_Analog_Validator <<<
END_FUNCTION_BLOCK

(* ---- FB_BlackBox_Recorder.st ---- *)
FUNCTION_BLOCK FB_BlackBox_Recorder
VAR_INPUT
    VI_Current_Data : ST_BlackBox_Record;
    VI_Freeze       : BOOL;
    VI_Reset        : BOOL;
END_VAR
VAR_OUTPUT
    VO_Frozen       : BOOL;
    VO_Records_Count: INT;
END_VAR
VAR
    L_Write_Index   : INT := 0;
    L_Initialized   : BOOL := FALSE;
END_VAR

IF NOT L_Initialized THEN
    L_Write_Index := GVL_Retain.G_BlackBox_LastIndex;
    IF L_Write_Index < 0 OR L_Write_Index >= GVL_CONSTANTS.C_MAX_BLACKBOX_RECORDS THEN
        L_Write_Index := 0;
        GVL_Retain.G_BlackBox_LastIndex := 0;
    END_IF;
    L_Initialized := TRUE;
END_IF;

IF VI_Reset THEN
    GVL_Retain.G_BlackBox_Frozen := FALSE;
END_IF;

IF VI_Freeze THEN
    GVL_Retain.G_BlackBox_Frozen := TRUE;
END_IF;

VO_Frozen := GVL_Retain.G_BlackBox_Frozen;

IF NOT GVL_Retain.G_BlackBox_Frozen THEN
    GVL_Retain.G_BlackBox_Buffer[L_Write_Index] := VI_Current_Data;
    GVL_Retain.G_BlackBox_LastIndex := L_Write_Index;

    L_Write_Index := L_Write_Index + 1;
    IF L_Write_Index >= GVL_CONSTANTS.C_MAX_BLACKBOX_RECORDS THEN
        L_Write_Index := 0;
    END_IF;
END_IF;

VO_Records_Count := GVL_CONSTANTS.C_MAX_BLACKBOX_RECORDS;
// >>> BULK_SYNC_ANCHOR: FB_BlackBox_Recorder <<<
END_FUNCTION_BLOCK

(* ---- FB_Config_Simulation.st ---- *)
// ==============================================================================
// Config simulation / validation function block
// Service/commissioning validation utility.
// Does NOT own runtime control and does NOT participate in heating phase runtime.
// ==============================================================================
FUNCTION_BLOCK FB_Config_Simulation
VAR_INPUT
    VI_Enable : BOOL;
    VI_Request : BOOL;
    VI_Confirm : BOOL;
END_VAR
VAR_OUTPUT
    VO_Executed : BOOL;
    VO_Result_OK : BOOL;
    VO_Error_Text : STRING(200);
END_VAR
VAR
    L_Error : BOOL;
END_VAR

VO_Executed := FALSE;
VO_Result_OK := GVL_CONFIG_SIMULATION.G_Simulation_Result_OK;
VO_Error_Text := GVL_CONFIG_SIMULATION.G_Simulation_Error_Text;

IF NOT VI_Enable THEN
    RETURN;
END_IF;

IF VI_Request AND VI_Confirm THEN

    L_Error := FALSE;
    VO_Result_OK := TRUE;
    VO_Error_Text := '';

    // Simulate INPUT constraints
    IF (GVL_CONFIG_CONTROL.STG_Reputation_Learning_Rate < 0.0) OR (GVL_CONFIG_CONTROL.STG_Reputation_Learning_Rate > 1.0) THEN
        VO_Result_OK := FALSE;
        VO_Error_Text := 'Invalid learning rate';
        L_Error := TRUE;
    END_IF;

    // Simulate SCENARIO logic
    IF GVL_CONFIG_CONTROL.STG_Night_Start_Hour = GVL_CONFIG_CONTROL.STG_Night_End_Hour THEN
        VO_Result_OK := FALSE;
        VO_Error_Text := 'Night window invalid';
        L_Error := TRUE;
    END_IF;

    // Simulate SAFETY
    IF GVL_CONFIG_CONTROL.STG_Stabilization_Delay_MS < 1000 THEN
        VO_Result_OK := FALSE;
        VO_Error_Text := 'Recovery delay too small';
        L_Error := TRUE;
    END_IF;

    // Simulate FAIL-SAFE policy
    IF NOT (
        GVL_CONFIG_CONTROL.STG_PLC_Inactive_Close_Gas OR
        GVL_CONFIG_CONTROL.STG_PLC_Inactive_Stop_Boiler OR
        GVL_CONFIG_CONTROL.STG_PLC_Inactive_Block_Heating OR
        GVL_CONFIG_CONTROL.STG_PLC_Inactive_Stop_Vent OR
        GVL_CONFIG_CONTROL.STG_PLC_Inactive_Block_Water
    ) THEN
        VO_Result_OK := FALSE;
        VO_Error_Text := 'Fail-safe disabled';
        L_Error := TRUE;
    END_IF;

    GVL_CONFIG_SIMULATION.G_Simulation_Result_OK := NOT L_Error;
    GVL_CONFIG_SIMULATION.G_Simulation_Error_Text := VO_Error_Text;
    GVL_CONFIG_SIMULATION.G_Simulation_Last_Run_MS := GVL_TIME_SERVICE.G_Now_MS;
    VO_Executed := TRUE;

END_IF;

END_FUNCTION_BLOCK
// >>> BULK_SYNC_ANCHOR: FB_Config_Simulation <<<

(* ---- FB_Distributed_Authority_Arbitration.st ---- *)
FUNCTION_BLOCK FB_Distributed_Authority_Arbitration
VAR_INPUT
    VI_Enable : BOOL;
    VI_System_Time_MS : UDINT;
END_VAR
VAR
    L_State : ST_Distributed_Authority_State;
    L_Lease_Expired : BOOL;

    L_Finalized_Runtime_Continuity : BOOL;
END_VAR

IF NOT VI_Enable THEN
    GVL_Distributed_Authority.G_Runtime_Valid := FALSE;
    RETURN;
END_IF;

L_State.Runtime_Valid := TRUE;
L_State.Runtime_System_Time_MS := VI_System_Time_MS;

L_State.Controller_Id :=
    GVL_Distributed_Runtime.G_Local_Node_State.Controller_Id;

L_State.Runtime_Node_Id :=
    GVL_Distributed_Runtime.G_Local_Node_State.Runtime_Node_Id;

L_State.Authority_Domain_Id :=
    GVL_Distributed_Runtime.G_Local_Node_State.Authority_Domain_Id;

L_State.Authority_Election_Active := TRUE;

L_Lease_Expired :=
    (VI_System_Time_MS - GVL_Distributed_Authority.G_Authority_Lease_Start_MS)
    > GVL_Distributed_Authority.G_Authority_Lease_Duration_MS;

L_State.Authority_Lease_Expired := L_Lease_Expired;
L_State.Authority_Lease_Valid := NOT L_Lease_Expired;

L_State.Replication_Consensus_Healthy :=
    GVL_Distributed_Runtime.G_Distributed_Replication_Healthy;

L_State.Replication_Consensus_Stale :=
    NOT GVL_Distributed_Runtime.G_Distributed_Replication_Healthy;

L_Finalized_Runtime_Continuity :=
    GVL_SEMANTIC_PROGRESS.Semantic_Forward_Progress_Valid
    AND GVL_SEMANTIC_PROGRESS.Semantic_Execution_Continuity_OK
    AND NOT GVL_SEMANTIC_PROGRESS.Semantic_Progress_Lease_Expired
    AND NOT GVL_SEMANTIC_PROGRESS.Semantic_Progress_Quarantine_Active
    AND GVL_RUNTIME_SNAPSHOT.Snapshot_Frozen
    AND GVL_RUNTIME_SNAPSHOT.Snapshot_Publication_Allowed
    AND GVL_RUNTIME_SNAPSHOT.Snapshot_Copy_Valid
    AND GVL_RUNTIME_SNAPSHOT.Snapshot_Isolation_Valid
    AND NOT GVL_RUNTIME_SNAPSHOT.Snapshot_Mutation_Detected
    AND GVL_DISTRIBUTED_SNAPSHOT.Distributed_Publication_Reconciled
    AND GVL_DISTRIBUTED_SNAPSHOT.Distributed_Publication_Freeze_Valid
    AND GVL_DISTRIBUTED_SNAPSHOT.Distributed_Snapshot_Consistent
    AND GVL_DISTRIBUTED_COMMIT.Distributed_Commit_Valid
    AND GVL_DISTRIBUTED_COMMIT.Publication_Prepare_Valid
    AND GVL_DISTRIBUTED_COMMIT.Publication_Commit_Confirmed
    AND NOT GVL_DISTRIBUTED_COMMIT.Peer_Commit_Mismatch
    AND NOT GVL_DISTRIBUTED_COMMIT.Commit_Lease_Expired
    AND GVL_OUTPUT_EPOCH.Output_Publication_Valid
    AND GVL_OUTPUT_EPOCH.Output_Runtime_Epoch_Valid
    AND NOT GVL_OUTPUT_EPOCH.Output_Lease_Expired
    AND NOT GVL_OUTPUT_EPOCH.Output_Forced_Safe_Decay
    AND GVL_COMMAND_VERIFY.PreOutput_Barrier_OK
    AND NOT GVL_COMMAND_VERIFY.PreOutput_Block_IO;

L_State.Distributed_Safety_Barrier_OK :=
    GVL_Runtime_Restart_Continuity.G_Runtime_Valid
    AND NOT GVL_Config_Activation.G_Config_Quarantine_Active
    AND NOT GVL_Distributed_Runtime.G_Split_Brain_Suspected
    AND GVL_IO_Binding_Runtime.G_Runtime_Valid
    AND L_Finalized_Runtime_Continuity;

IF NOT L_State.Distributed_Safety_Barrier_OK THEN

    L_State.Split_Brain_Blocked := TRUE;
    L_State.Authority_Observer_Only := TRUE;

    L_State.Status_Code := 3;
    L_State.Status_Text :=
        'Distributed authority blocked by safety barrier';

ELSIF L_State.Replication_Consensus_Healthy
   AND NOT L_Lease_Expired
   AND L_Finalized_Runtime_Continuity THEN

    L_State.Authority_Master_Elected := TRUE;

    L_State.Recovery_Authority_Allowed := TRUE;
    L_State.Rollback_Authority_Allowed := TRUE;
    L_State.Quarantine_Authority_Allowed := TRUE;

    L_State.Status_Code := 1;
    L_State.Status_Text :=
        'Distributed master authority active';

ELSE

    L_State.Authority_Backup_Elected := TRUE;

    L_State.Status_Code := 2;
    L_State.Status_Text :=
        'Distributed backup authority active';

END_IF;

GVL_Distributed_Authority.G_Authority_State := L_State;

GVL_Distributed_Authority.G_Split_Brain_Blocked :=
    L_State.Split_Brain_Blocked;

GVL_Distributed_Authority.G_Distributed_Safety_Barrier_OK :=
    L_State.Distributed_Safety_Barrier_OK;

GVL_Distributed_Authority.G_Runtime_Valid := TRUE;
GVL_Distributed_Authority.G_Last_Update_MS := VI_System_Time_MS;
GVL_Distributed_Authority.G_Status_Code := L_State.Status_Code;
GVL_Distributed_Authority.G_Status_Text := L_State.Status_Text;

END_FUNCTION_BLOCK

(* ---- FB_Distributed_Recovery_Lock_Runtime.st ---- *)
FUNCTION_BLOCK FB_Distributed_Recovery_Lock_Runtime
VAR_INPUT
    VI_Enable : BOOL;
    VI_System_Time_MS : UDINT;
END_VAR
VAR
    L_Lock : ST_Distributed_Recovery_Lock;
    L_Finalized_Runtime_Continuity : BOOL;
END_VAR

IF NOT VI_Enable THEN
    GVL_Distributed_Recovery_Lock.G_Runtime_Valid := FALSE;
    RETURN;
END_IF;

L_Lock := GVL_Distributed_Recovery_Lock.G_Recovery_Lock;

L_Lock.Runtime_System_Time_MS := VI_System_Time_MS;
L_Lock.Lock_Valid := TRUE;

// Finalized runtime continuity proof chain.
L_Finalized_Runtime_Continuity :=
    GVL_SEMANTIC_PROGRESS.Semantic_Forward_Progress_Valid
    AND GVL_SEMANTIC_PROGRESS.Semantic_Execution_Continuity_OK
    AND NOT GVL_SEMANTIC_PROGRESS.Semantic_Progress_Lease_Expired
    AND NOT GVL_SEMANTIC_PROGRESS.Semantic_Progress_Quarantine_Active
    AND GVL_RUNTIME_SNAPSHOT.Snapshot_Frozen
    AND GVL_RUNTIME_SNAPSHOT.Snapshot_Publication_Allowed
    AND GVL_RUNTIME_SNAPSHOT.Snapshot_Copy_Valid
    AND GVL_RUNTIME_SNAPSHOT.Snapshot_Isolation_Valid
    AND NOT GVL_RUNTIME_SNAPSHOT.Snapshot_Mutation_Detected
    AND GVL_DISTRIBUTED_SNAPSHOT.Distributed_Publication_Reconciled
    AND GVL_DISTRIBUTED_SNAPSHOT.Distributed_Publication_Freeze_Valid
    AND GVL_DISTRIBUTED_SNAPSHOT.Distributed_Snapshot_Consistent
    AND GVL_DISTRIBUTED_COMMIT.Distributed_Commit_Valid
    AND GVL_DISTRIBUTED_COMMIT.Publication_Prepare_Valid
    AND GVL_DISTRIBUTED_COMMIT.Publication_Commit_Confirmed
    AND NOT GVL_DISTRIBUTED_COMMIT.Peer_Commit_Mismatch
    AND NOT GVL_DISTRIBUTED_COMMIT.Commit_Lease_Expired
    AND GVL_OUTPUT_EPOCH.Output_Publication_Valid
    AND GVL_OUTPUT_EPOCH.Output_Runtime_Epoch_Valid
    AND NOT GVL_OUTPUT_EPOCH.Output_Lease_Expired
    AND NOT GVL_OUTPUT_EPOCH.Output_Forced_Safe_Decay
    AND GVL_COMMAND_VERIFY.PreOutput_Barrier_OK
    AND NOT GVL_COMMAND_VERIFY.PreOutput_Block_IO;

// Cluster-exclusive recovery execution lock.
IF GVL_Distributed_Runtime.G_Split_Brain_Suspected
   OR GVL_Distributed_Projection_Ownership.G_Any_Ownership_Conflict
   OR GVL_Runtime_Sessions.G_Any_Stale_Session
   OR NOT L_Finalized_Runtime_Continuity THEN

    L_Lock.Lock_Conflict := TRUE;
    L_Lock.Distributed_Execution_Allowed := FALSE;

    GVL_Distributed_Recovery_Lock.G_Recovery_Execution_Blocked := TRUE;
    GVL_Distributed_Recovery_Lock.G_Rollback_Execution_Blocked := TRUE;
    GVL_Distributed_Recovery_Lock.G_Reopen_Execution_Blocked := TRUE;

    L_Lock.Status_Code := 3;
    L_Lock.Status_Text :=
        'Distributed recovery execution locked';

ELSE

    L_Lock.Recovery_Lock_Active := TRUE;
    L_Lock.Distributed_Execution_Allowed := TRUE;

    GVL_Distributed_Recovery_Lock.G_Recovery_Execution_Blocked := FALSE;
    GVL_Distributed_Recovery_Lock.G_Rollback_Execution_Blocked := FALSE;
    GVL_Distributed_Recovery_Lock.G_Reopen_Execution_Blocked := FALSE;

    L_Lock.Status_Code := 0;
    L_Lock.Status_Text :=
        'Distributed recovery lock healthy';

END_IF;

GVL_Distributed_Recovery_Lock.G_Recovery_Lock := L_Lock;

GVL_Distributed_Recovery_Lock.G_Runtime_Valid := TRUE;
GVL_Distributed_Recovery_Lock.G_Last_Update_MS :=
    VI_System_Time_MS;

GVL_Distributed_Recovery_Lock.G_Status_Code :=
    L_Lock.Status_Code;

GVL_Distributed_Recovery_Lock.G_Status_Text :=
    L_Lock.Status_Text;

END_FUNCTION_BLOCK

(* ---- FB_FloorHeating_Controller.st ---- *)
FUNCTION_BLOCK FB_FloorHeating_Controller
VAR_INPUT
    VI_Current_Temp : REAL;
    VI_Config : ST_FloorHeating_Circuit_Config;
    VI_Tariff : ST_Tariff_Config;
    VI_Current_Hour : UINT;
    VI_IsActivePLC : BOOL;
    VI_System_Time_MS : UDINT;
END_VAR
VAR_OUTPUT
    VO_Pump_Run : BOOL;
    VO_Valve_Pos : REAL; // 0..100%
    VO_Valve_Bool : BOOL; // ШИМ выход для термоэлектрического привода
    VO_Effective_Setpoint : REAL;
END_VAR
VAR
    L_Is_Night : BOOL;
    L_PID : FB_PID_Controller;
    L_Last_Time : UDINT;
    L_Cycle_Time_S : REAL;
    L_PWM_Period_MS : UDINT;
    L_PWM_Duty_MS : UDINT;
    L_Current_Phase_MS : UDINT;
    L_PWM_Start_Time : UDINT;
END_VAR

// Вычисление времени цикла
IF L_Last_Time = 0 THEN
    L_Last_Time := VI_System_Time_MS;
    L_Cycle_Time_S := 1.0;
ELSE
    L_Cycle_Time_S := UDINT_TO_REAL((SEL(VI_System_Time_MS >= L_Last_Time, VI_System_Time_MS - L_Last_Time, (4294967295 - L_Last_Time) + VI_System_Time_MS + 1))) / 1000.0;
    L_Last_Time := VI_System_Time_MS;
END_IF;
IF L_Cycle_Time_S <= 0.0 THEN L_Cycle_Time_S := 0.01; END_IF;

// 1. Определение активного тарифа
IF VI_Tariff.Enabled THEN
    IF VI_Tariff.Night_Start_Hour > VI_Tariff.Night_End_Hour THEN
        // Переход через полночь (например, 23:00 - 07:00)
        L_Is_Night := (VI_Current_Hour >= VI_Tariff.Night_Start_Hour) OR (VI_Current_Hour < VI_Tariff.Night_End_Hour);
    ELSE
        // В пределах одного дня
        L_Is_Night := (VI_Current_Hour >= VI_Tariff.Night_Start_Hour) AND (VI_Current_Hour < VI_Tariff.Night_End_Hour);
    END_IF;
ELSE
    L_Is_Night := FALSE;
END_IF;

// 2. Расчет эффективной уставки
VO_Effective_Setpoint := VI_Config.design_temp;
IF L_Is_Night THEN
    VO_Effective_Setpoint := VO_Effective_Setpoint + VI_Tariff.Boost_Delta;
END_IF;

// 3. ПИД-регулирование
L_PID(
    VI_SetPoint := VO_Effective_Setpoint,
    VI_ProcessValue := VI_Current_Temp,
    VI_Kp := VI_Config.pid_kp,
    VI_Tn := 300.0,
    VI_Tv := 0.0,
    VI_Y_Min := 0.0,
    VI_Y_Max := 100.0,
    VI_Cycle_Time_S := L_Cycle_Time_S,
    VO_Output => VO_Valve_Pos
);

// 4. ШИМ-модуляция для термоэлектрического привода
IF VI_Config.pwm_period_s > 0 THEN
    L_PWM_Period_MS := TO_UDINT(VI_Config.pwm_period_s) * 1000;
ELSE
    L_PWM_Period_MS := 600000; // 10 минут
END_IF;

L_Current_Phase_MS := (SEL(VI_System_Time_MS >= L_PWM_Start_Time, VI_System_Time_MS - L_PWM_Start_Time, (4294967295 - L_PWM_Start_Time) + VI_System_Time_MS + 1));
IF L_Current_Phase_MS >= L_PWM_Period_MS THEN
    L_PWM_Start_Time := VI_System_Time_MS - (L_Current_Phase_MS - L_PWM_Period_MS); // Сохраняем остаток для точности
    L_Current_Phase_MS := (SEL(VI_System_Time_MS >= L_PWM_Start_Time, VI_System_Time_MS - L_PWM_Start_Time, (4294967295 - L_PWM_Start_Time) + VI_System_Time_MS + 1));
END_IF;

L_PWM_Duty_MS := TO_UDINT((VO_Valve_Pos / 100.0) * TO_REAL(L_PWM_Period_MS));

IF VI_IsActivePLC THEN
    VO_Pump_Run := (VO_Valve_Pos > 5.0);

    IF VO_Valve_Pos >= 100.0 THEN
        VO_Valve_Bool := TRUE;
    ELSIF VO_Valve_Pos <= 0.0 THEN
        VO_Valve_Bool := FALSE;
    ELSE
        VO_Valve_Bool := (L_Current_Phase_MS <= L_PWM_Duty_MS);
    END_IF;
ELSE
    VO_Pump_Run := FALSE;
    VO_Valve_Bool := FALSE;
END_IF;
END_FUNCTION_BLOCK

(* ---- FB_Gateway_Interface.st ---- *)
FUNCTION_BLOCK FB_Gateway_Interface
VAR_INPUT
    VI_System_Time_MS           : UDINT;
    VI_Local_PLC_Role           : E_PLC_ROLE;
    VI_Incoming_Command         : ST_Gateway_Command;
    VI_Command_Received         : BOOL;
    VI_Outdoor_Temp             : REAL;
    VI_Security_Armed           : BOOL;
    VI_Flood_Alarm_Active       : BOOL;
    VI_Gas_Alarm_Active         : BOOL;
    VI_Fire_Alarm_Active        : BOOL;
    VI_Methane_Concentration    : REAL;
    VI_Active_Scenario          : E_SCENARIO_TYPE;
    VI_Send_2FA_Req             : BOOL;
    VI_2FA_Code                 : STRING(6);
END_VAR

VAR_IN_OUT
    VI_FloorHeating_Temps       : ARRAY[1..GVL_CONSTANTS.C_MAX_HEATING_CIRCUITS] OF REAL;
    VI_Room_Temps               : ARRAY[1..GVL_CONSTANTS.C_MAX_ZONES] OF REAL;
    VI_Zone_Valve_States        : ARRAY[1..GVL_CONSTANTS.C_MAX_HEATING_CIRCUITS] OF BOOL;
    VI_Manifold_Pressures       : ARRAY[1..GVL_CONSTANTS.C_MAX_MANIFOLDS] OF REAL;
    VI_Manifold_Pump_States     : ARRAY[1..GVL_CONSTANTS.C_MAX_MANIFOLDS] OF BOOL;
    VI_Lighting_Base_Levels     : ARRAY[1..GVL_CONSTANTS.C_MAX_LIGHT_ZONES] OF BYTE;
    VI_Socket_States            : ARRAY[1..GVL_CONSTANTS.C_MAX_SOCKETS] OF BOOL;
    VI_Blinds_Positions         : ARRAY[1..GVL_CONSTANTS.C_MAX_BLINDS] OF BYTE;
    VI_Allowed_IPs              : ARRAY[1..GVL_CONSTANTS.C_MAX_ALLOWED_IPS] OF STRING(15);
END_VAR

VAR_OUTPUT
    VO_Modbus_Registers         : ARRAY[0..GVL_CONSTANTS.C_MAX_MODBUS_REGISTERS-1] OF WORD;
    VO_Lighting_Override        : ARRAY[1..GVL_CONSTANTS.C_MAX_LIGHT_ZONES] OF BYTE;
    VO_Blinds_Override          : ARRAY[1..GVL_CONSTANTS.C_MAX_BLINDS] OF BYTE;
    VO_Socket_Override          : ARRAY[1..GVL_CONSTANTS.C_MAX_SOCKETS] OF BOOL;
    VO_Arm_Req                  : BOOL;
    VO_Disarm_Req               : BOOL;
    VO_PIN_Code                 : STRING(4);
    VO_RFID_Tag                 : STRING(20);
    VO_2FA_Code_In              : STRING(6);
    VO_Data_Ready               : BOOL;
    VO_HMI_Status_Message       : STRING(200);
    VO_Telegram_Msg             : STRING(200);
    VO_Send_Telegram            : BOOL;
    VO_Set_Scenario_Req         : BOOL;
    VO_Target_Scenario          : E_SCENARIO_TYPE;
    VO_Set_Temp_Req             : BOOL;
    VO_Target_Zone              : INT;
    VO_Target_Temp              : REAL;
    VO_Set_Vent_Req             : BOOL;
    VO_Target_Vent_Speed        : BYTE;
    VO_Reset_Errors_Req         : BOOL;
    VO_Set_Config_Req           : BOOL;
    VO_Sync_Time_Req            : BOOL;
    VO_New_Time_MS              : UDINT;
END_VAR

VAR
    L_last_update_time          : UDINT;
    L_i                         : INT;
    L_j                         : INT;
    L_idx                       : INT;
    L_tmp_word                  : WORD;
    L_Code_UDINT                : UDINT;
    L_Prev_Fire                 : BOOL;
    L_Prev_Gas                  : BOOL;
    L_Prev_Flood                : BOOL;
    L_Prev_Security             : BOOL;
    L_Deduplicator              : FB_Command_Deduplication;
    L_IP_Allowed                : BOOL;
    L_Process_Command           : ST_Gateway_Command;
    L_Has_Command_To_Process    : BOOL;
END_VAR

VAR RETAIN
    L_Command_Buffer            : ARRAY[1..GVL_CONSTANTS.C_MAX_GATEWAY_COMMANDS] OF ST_Gateway_Command;
    L_Buffer_Head               : INT := 1;
    L_Buffer_Tail               : INT := 1;
    L_Buffer_Count              : INT := 0;
END_VAR

VO_Send_Telegram := FALSE;
IF VI_Fire_Alarm_Active AND NOT L_Prev_Fire THEN
    VO_Telegram_Msg := 'ВНИМАНИЕ! ПОЖАРНАЯ ТРЕВОГА!';
    VO_Send_Telegram := TRUE;
END_IF;
IF VI_Gas_Alarm_Active AND NOT L_Prev_Gas THEN
    VO_Telegram_Msg := 'ВНИМАНИЕ! УТЕЧКА ГАЗА!';
    VO_Send_Telegram := TRUE;
END_IF;
IF VI_Flood_Alarm_Active AND NOT L_Prev_Flood THEN
    VO_Telegram_Msg := 'ВНИМАНИЕ! ПРОТЕЧКА ВОДЫ!';
    VO_Send_Telegram := TRUE;
END_IF;
IF VI_Security_Armed AND NOT L_Prev_Security THEN
    VO_Telegram_Msg := 'ОХРАНА ВКЛЮЧЕНА';
    VO_Send_Telegram := TRUE;
ELSIF NOT VI_Security_Armed AND L_Prev_Security THEN
    VO_Telegram_Msg := 'ОХРАНА ОТКЛЮЧЕНА';
    VO_Send_Telegram := TRUE;
END_IF;

L_Prev_Fire := VI_Fire_Alarm_Active;
L_Prev_Gas := VI_Gas_Alarm_Active;
L_Prev_Flood := VI_Flood_Alarm_Active;
L_Prev_Security := VI_Security_Armed;

IF (VI_System_Time_MS - L_last_update_time) >= GVL_CONSTANTS.C_MS_IN_SECOND THEN
    L_last_update_time := VI_System_Time_MS;
    L_tmp_word := 0;
    IF VI_Local_PLC_Role = E_PLC_ROLE.ROLE_ACTIVE THEN L_tmp_word := L_tmp_word OR 1; END_IF;
    IF VI_Security_Armed THEN L_tmp_word := L_tmp_word OR 2; END_IF;
    IF VI_Flood_Alarm_Active THEN L_tmp_word := L_tmp_word OR 4; END_IF;
    IF VI_Gas_Alarm_Active THEN L_tmp_word := L_tmp_word OR 8; END_IF;
    IF VI_Fire_Alarm_Active THEN L_tmp_word := L_tmp_word OR 16; END_IF;
    VO_Modbus_Registers[0] := L_tmp_word;

    FOR L_i := 1 TO GVL_CONSTANTS.C_MAX_HEATING_CIRCUITS DO
        VO_Modbus_Registers[L_i] := TO_WORD(TO_INT(VI_FloorHeating_Temps[L_i] * REAL#10.0));
    END_FOR;

    FOR L_i := 1 TO GVL_CONSTANTS.C_MAX_ZONES DO
        VO_Modbus_Registers[16 + L_i] := TO_WORD(TO_INT(VI_Room_Temps[L_i] * REAL#10.0));
    END_FOR;

    L_tmp_word := 0;
    FOR L_i := 1 TO GVL_CONSTANTS.C_MAX_HEATING_CIRCUITS DO
        IF VI_Zone_Valve_States[L_i] THEN
            L_tmp_word := L_tmp_word OR SHL(TO_WORD(1), L_i - 1);
        END_IF;
    END_FOR;
    VO_Modbus_Registers[33] := L_tmp_word;

    FOR L_i := 1 TO GVL_CONSTANTS.C_MAX_MANIFOLDS DO
        VO_Modbus_Registers[33 + L_i] := TO_WORD(TO_INT(VI_Manifold_Pressures[L_i] * REAL#100.0));
    END_FOR;

    FOR L_i := 1 TO GVL_CONSTANTS.C_MAX_LIGHT_ZONES DO
        VO_Modbus_Registers[39 + L_i] := TO_WORD(VI_Lighting_Base_Levels[L_i]);
    END_FOR;

    FOR L_i := 1 TO GVL_CONSTANTS.C_MAX_BLINDS DO
        VO_Modbus_Registers[71 + L_i] := TO_WORD(VI_Blinds_Positions[L_i]);
    END_FOR;

    FOR L_i := 0 TO (GVL_CONSTANTS.C_MAX_SOCKETS - 1) / 16 DO
        L_tmp_word := 0;
        FOR L_j := 1 TO 16 DO
            L_idx := (L_i * 16) + L_j;
            IF L_idx <= GVL_CONSTANTS.C_MAX_SOCKETS THEN
                IF VI_Socket_States[L_idx] THEN
                    L_tmp_word := L_tmp_word OR SHL(TO_WORD(1), L_j - 1);
                END_IF;
            END_IF;
        END_FOR;
        VO_Modbus_Registers[92 + L_i] := L_tmp_word;
    END_FOR;

    VO_Modbus_Registers[100] := SEL(VI_Send_2FA_Req, 0, 1);
    IF VI_Send_2FA_Req THEN
        L_Code_UDINT := STRING_TO_UDINT(VI_2FA_Code);
        VO_Modbus_Registers[101] := TO_WORD(L_Code_UDINT AND 16#FFFF);
        VO_Modbus_Registers[102] := TO_WORD(SHR(L_Code_UDINT, 16));
    ELSE
        VO_Modbus_Registers[101] := 0;
        VO_Modbus_Registers[102] := 0;
    END_IF;

    VO_Data_Ready := TRUE;
END_IF;

VO_Arm_Req := FALSE;
VO_Disarm_Req := FALSE;
VO_Set_Scenario_Req := FALSE;
VO_Set_Temp_Req := FALSE;
VO_Set_Vent_Req := FALSE;
VO_Reset_Errors_Req := FALSE;
VO_Set_Config_Req := FALSE;
VO_Sync_Time_Req := FALSE;
L_Has_Command_To_Process := FALSE;

IF VI_Command_Received THEN
    IF VI_Local_PLC_Role = E_PLC_ROLE.ROLE_ACTIVE THEN
        L_Process_Command := VI_Incoming_Command;
        L_Has_Command_To_Process := TRUE;
    ELSE
        IF L_Buffer_Count < GVL_CONSTANTS.C_MAX_GATEWAY_COMMANDS THEN
            L_Command_Buffer[L_Buffer_Head] := VI_Incoming_Command;
            L_Buffer_Head := L_Buffer_Head + 1;
            IF L_Buffer_Head > GVL_CONSTANTS.C_MAX_GATEWAY_COMMANDS THEN L_Buffer_Head := 1; END_IF;
            L_Buffer_Count := L_Buffer_Count + 1;
        END_IF;
    END_IF;
END_IF;

IF NOT L_Has_Command_To_Process AND (VI_Local_PLC_Role = E_PLC_ROLE.ROLE_ACTIVE) AND (L_Buffer_Count > 0) THEN
    L_Process_Command := L_Command_Buffer[L_Buffer_Tail];
    L_Buffer_Tail := L_Buffer_Tail + 1;
    IF L_Buffer_Tail > GVL_CONSTANTS.C_MAX_GATEWAY_COMMANDS THEN L_Buffer_Tail := 1; END_IF;
    L_Buffer_Count := L_Buffer_Count - 1;
    L_Has_Command_To_Process := TRUE;
END_IF;

IF L_Has_Command_To_Process THEN
    L_IP_Allowed := FALSE;
    IF L_Process_Command.source_ip = '' THEN
        L_IP_Allowed := TRUE;
    ELSE
        FOR L_i := 1 TO GVL_CONSTANTS.C_MAX_ALLOWED_IPS DO
            IF VI_Allowed_IPs[L_i] = L_Process_Command.source_ip THEN
                L_IP_Allowed := TRUE;
                EXIT;
            END_IF;
        END_FOR;
    END_IF;

    IF NOT L_IP_Allowed THEN
        VO_HMI_Status_Message := 'Gateway: Ошибка безопасности (Неизвестный IP)';
        RETURN;
    END_IF;

    IF L_Process_Command.crc32 <> DWORD#0 THEN
        VO_HMI_Status_Message := 'Gateway: CRC unsupported in legacy mode';
        RETURN;
    END_IF;

    L_Deduplicator(
        VI_Command_ID := L_Process_Command.command_id,
        VI_Command_Type := L_Process_Command.command_type,
        VI_Command_Value := L_Process_Command.target_value,
        VI_System_Time_MS := VI_System_Time_MS
    );

    IF L_Deduplicator.VO_Is_New_Command THEN
        CASE L_Process_Command.command_type OF
            E_Gateway_Command_Type.CMD_SET_SCENARIO:
                VO_Set_Scenario_Req := TRUE;
                VO_Target_Scenario := L_Process_Command.target_scenario;
                VO_HMI_Status_Message := 'Gateway: Сценарий изменен';
            E_Gateway_Command_Type.CMD_SET_LIGHT:
                IF (L_Process_Command.target_zone >= 1) AND (L_Process_Command.target_zone <= GVL_CONSTANTS.C_MAX_LIGHT_ZONES) THEN
                    VO_Lighting_Override[L_Process_Command.target_zone] := TO_BYTE(L_Process_Command.target_value);
                    VO_HMI_Status_Message := 'Gateway: Команда освещения принята';
                END_IF;
            E_Gateway_Command_Type.CMD_SET_BLINDS:
                IF (L_Process_Command.target_zone >= 1) AND (L_Process_Command.target_zone <= GVL_CONSTANTS.C_MAX_BLINDS) THEN
                    VO_Blinds_Override[L_Process_Command.target_zone] := TO_BYTE(L_Process_Command.target_value);
                    VO_HMI_Status_Message := 'Gateway: Команда штор принята';
                END_IF;
            E_Gateway_Command_Type.CMD_SET_SOCKET:
                IF (L_Process_Command.target_zone >= 1) AND (L_Process_Command.target_zone <= GVL_CONSTANTS.C_MAX_SOCKETS) THEN
                    VO_Socket_Override[L_Process_Command.target_zone] := L_Process_Command.target_on_off;
                    VO_HMI_Status_Message := 'Gateway: Команда розетки принята';
                END_IF;
            E_Gateway_Command_Type.CMD_SET_SECURITY:
                IF L_Process_Command.target_armed THEN VO_Arm_Req := TRUE; ELSE VO_Disarm_Req := TRUE; END_IF;
                VO_PIN_Code := L_Process_Command.target_pin;
                VO_2FA_Code_In := L_Process_Command.target_2fa_code;
                VO_HMI_Status_Message := 'Gateway: Запрос охраны принят';
            E_Gateway_Command_Type.CMD_SET_TEMP:
                IF (L_Process_Command.target_zone >= 1) AND (L_Process_Command.target_zone <= GVL_CONSTANTS.C_MAX_HEATING_CIRCUITS) THEN
                    VO_Set_Temp_Req := TRUE;
                    VO_Target_Zone := L_Process_Command.target_zone;
                    VO_Target_Temp := L_Process_Command.target_value;
                    VO_HMI_Status_Message := 'Gateway: Уставка температуры изменена';
                END_IF;
            E_Gateway_Command_Type.CMD_SET_VENT:
                VO_Set_Vent_Req := TRUE;
                VO_Target_Vent_Speed := TO_BYTE(L_Process_Command.target_value);
                VO_HMI_Status_Message := 'Gateway: Уставка вентиляции изменена';
            E_Gateway_Command_Type.CMD_TELEGRAM_MSG:
                VO_Telegram_Msg := L_Process_Command.telegram_msg;
                VO_Send_Telegram := TRUE;
                VO_HMI_Status_Message := 'Gateway: Сообщение Telegram отправлено';
            E_Gateway_Command_Type.CMD_SYNC_TIME:
                VO_Sync_Time_Req := TRUE;
                VO_New_Time_MS := REAL_TO_UDINT(L_Process_Command.target_value);
                VO_HMI_Status_Message := 'Gateway: Время синхронизировано';
            E_Gateway_Command_Type.CMD_RESET_ERRORS:
                VO_Reset_Errors_Req := TRUE;
                VO_HMI_Status_Message := 'Gateway: Запрос на сброс ошибок принят';
            E_Gateway_Command_Type.CMD_SET_CONFIG:
                VO_Set_Config_Req := TRUE;
                VO_HMI_Status_Message := 'Gateway: Запрос на применение конфигурации принят';
        END_CASE;
    ELSE
        VO_HMI_Status_Message := 'Gateway: duplicate command ignored';
    END_IF;
END_IF;

// >>> BULK_SYNC_ANCHOR: FB_Gateway_Interface <<<
END_FUNCTION_BLOCK

(* ---- FB_Heating_Circuit_Control.st ---- *)
// ==============================================================================
// Heating circuit control helper
//
// Internal refactoring helper for FB_Heating_System_Manager.
// Owns per-circuit sensor validation, temperature source fallback,
// floor-heating controller call, overheat shutdown, and rule action projection.
//
// Temperature source selection is confidence-aware:
// - range invalid still blocks that source;
// - passive input-quality confidence can prefer a healthier fallback;
// - degraded-but-range-valid sources remain operational if no better source exists.
//
// Publishes only canonical runtime projection semantics to
// GVL_Heating_Runtime_Projection. Explainability, predictive observation and
// supervisory ingestion consume that projection downstream.
// ==============================================================================
FUNCTION_BLOCK FB_Heating_Circuit_Control
VAR_INPUT
    VI_System_Time_MS : UDINT;
    VI_Current_Hour : UINT;
    VI_IsActivePLC : BOOL;
    VI_Config : ST_Heating_Config;
    VI_Tariff : ST_Tariff_Config;
    VI_Scenario_Adjust : REAL;
END_VAR

VAR_IN_OUT
    VI_Zone_Configs : ARRAY[1..GVL_CONSTANTS.C_MAX_HEATING_CIRCUITS] OF ST_FloorHeating_Circuit_Config;
    VI_Floor_Temps : ARRAY[1..GVL_CONSTANTS.C_MAX_HEATING_CIRCUITS] OF REAL;
    VI_Room_Temps : ARRAY[1..16] OF REAL;
    VI_Rule_Actions : ARRAY[1..GVL_CONSTANTS.C_MAX_RULES] OF ST_Rule_Action;
END_VAR

VAR_OUTPUT
    VO_Zone_Valves : ARRAY[1..GVL_CONSTANTS.C_MAX_HEATING_CIRCUITS] OF BOOL;
    VO_Heating_Sensor_Fault : BOOL;
END_VAR

VAR
    L_i : INT;
    L_j : INT;
    L_Climate_Zone_ID : INT;
    L_Zone_Config : ST_FloorHeating_Circuit_Config;
    L_Current_Temp : REAL;
    L_Sensor_Error : BOOL;
    L_Floor_Source_Valid : BOOL;
    L_Room_Source_Valid : BOOL;
    L_Floor_Confidence : REAL;
    L_Room_Confidence : REAL;
    L_Min_Source_Confidence : REAL;
    L_Primary_Source_Code : UINT;
    L_Selected_Source_Code : UINT;
    L_Primary_Confidence : REAL;
    L_Fallback_Confidence : REAL;
    L_Selected_Confidence : REAL;
    L_Fallback_Active : BOOL;
    L_Source_Degraded : BOOL;
    L_Reason_Code : UINT;
    L_Reason_Text : STRING(128);
    L_Selected_Source_Text : STRING(64);
    L_Comfort_Target : REAL;
    L_Economy_Target : REAL;
    L_Long_Away_Target : REAL;
    L_Effective_Target : REAL;
    L_Max_Target : REAL;

    L_Prev_Selected_Source_Code : ARRAY[1..GVL_CONSTANTS.C_MAX_HEATING_CIRCUITS] OF UINT;
    L_Prev_Fallback_Active : ARRAY[1..GVL_CONSTANTS.C_MAX_HEATING_CIRCUITS] OF BOOL;
    L_Prev_Source_Loss : ARRAY[1..GVL_CONSTANTS.C_MAX_HEATING_CIRCUITS] OF BOOL;
    L_Source_Loss_Active : BOOL;

    L_Source_Switched_Event : BOOL;
    L_Fallback_Activated_Event : BOOL;
    L_Fallback_Recovered_Event : BOOL;
    L_Source_Loss_Event : BOOL;
    L_Last_Event_Code : UINT;
    L_Last_Event_Text : STRING(128);

    L_Floor_Controllers : ARRAY[1..GVL_CONSTANTS.C_MAX_HEATING_CIRCUITS] OF FB_FloorHeating_Controller;
    L_Overheat_Timer : ARRAY[1..GVL_CONSTANTS.C_MAX_HEATING_CIRCUITS] OF FB_System_Timer;
    fbFloorTempValidator : ARRAY[1..GVL_CONSTANTS.C_MAX_HEATING_CIRCUITS] OF FB_Analog_Validator;
    fbRoomTempValidator : ARRAY[1..16] OF FB_Analog_Validator;
END_VAR

VO_Heating_Sensor_Fault := FALSE;
L_Min_Source_Confidence := GVL_INPUT_VALIDATION_CONFIG.G_Min_Sensor_Confidence;

FOR L_i := 1 TO GVL_CONSTANTS.C_MAX_HEATING_CIRCUITS DO
    fbFloorTempValidator[L_i](
        VI_Value := VI_Floor_Temps[L_i],
        VI_Min_Valid := -40.0,
        VI_Max_Valid := 120.0,
        VI_Fallback_Mode := 0
    );

    L_Climate_Zone_ID := VI_Zone_Configs[L_i].zone;
    IF L_Climate_Zone_ID >= 1 AND L_Climate_Zone_ID <= 16 THEN
        fbRoomTempValidator[L_Climate_Zone_ID](
            VI_Value := VI_Room_Temps[L_Climate_Zone_ID],
            VI_Min_Valid := -40.0,
            VI_Max_Valid := 120.0,
            VI_Fallback_Mode := 0
        );
    END_IF;

    L_Floor_Source_Valid := NOT fbFloorTempValidator[L_i].VO_Error;
    L_Room_Source_Valid :=
        (L_Climate_Zone_ID >= 1) AND
        (L_Climate_Zone_ID <= 16) AND
        (NOT fbRoomTempValidator[L_Climate_Zone_ID].VO_Error);

    L_Floor_Confidence := REAL#1.0;
    IF GVL_INPUT_QUALITY.G_Floor_Temp_Quality[L_i].Quality_Visible THEN
        L_Floor_Confidence := GVL_INPUT_QUALITY.G_Floor_Temp_Quality[L_i].Confidence;
    END_IF;

    L_Room_Confidence := REAL#1.0;
    IF (L_Climate_Zone_ID >= 1) AND (L_Climate_Zone_ID <= 16) THEN
        IF GVL_INPUT_QUALITY.G_Room_Temp_Quality[L_Climate_Zone_ID].Quality_Visible THEN
            L_Room_Confidence := GVL_INPUT_QUALITY.G_Room_Temp_Quality[L_Climate_Zone_ID].Confidence;
        END_IF;
    END_IF;

    IF L_Floor_Confidence < REAL#0.0 THEN
        L_Floor_Confidence := REAL#0.0;
    ELSIF L_Floor_Confidence > REAL#1.0 THEN
        L_Floor_Confidence := REAL#1.0;
    END_IF;

    IF L_Room_Confidence < REAL#0.0 THEN
        L_Room_Confidence := REAL#0.0;
    ELSIF L_Room_Confidence > REAL#1.0 THEN
        L_Room_Confidence := REAL#1.0;
    END_IF;

    // Floor overheat protection remains floor-bound and range-validity based.
    L_Overheat_Timer[L_i](
        IN := L_Floor_Source_Valid AND (fbFloorTempValidator[L_i].VO_Value > VI_Config.Overheat_Threshold),
        PT := T#60s,
        VI_System_Time_MS := VI_System_Time_MS
    );

    L_Current_Temp := REAL#0.0;
    L_Sensor_Error := FALSE;
    L_Selected_Source_Code := 0;
    L_Selected_Source_Text := 'none';
    L_Selected_Confidence := REAL#0.0;
    L_Fallback_Active := FALSE;
    L_Source_Degraded := FALSE;
    L_Reason_Code := 0;
    L_Reason_Text := 'OK';

    IF VI_Zone_Configs[L_i].control_type = 1 OR VI_Zone_Configs[L_i].control_type = 2 THEN
        L_Primary_Source_Code := 1; // room
        L_Primary_Confidence := L_Room_Confidence;
        L_Fallback_Confidence := L_Floor_Confidence;

        // Primary: room air temperature. If room quality is degraded and floor
        // source is healthier, prefer floor fallback without declaring hard fault.
        IF L_Room_Source_Valid AND
           ((L_Room_Confidence >= L_Min_Source_Confidence) OR NOT L_Floor_Source_Valid OR (L_Room_Confidence >= L_Floor_Confidence)) THEN
            L_Current_Temp := fbRoomTempValidator[L_Climate_Zone_ID].VO_Value;
            L_Selected_Source_Code := 1;
            L_Selected_Source_Text := 'room';
            L_Selected_Confidence := L_Room_Confidence;
        ELSIF L_Floor_Source_Valid THEN
            L_Current_Temp := fbFloorTempValidator[L_i].VO_Value;
            L_Selected_Source_Code := 2;
            L_Selected_Source_Text := 'floor';
            L_Selected_Confidence := L_Floor_Confidence;
            L_Fallback_Active := TRUE;
        ELSIF L_Room_Source_Valid THEN
            L_Current_Temp := fbRoomTempValidator[L_Climate_Zone_ID].VO_Value;
            L_Selected_Source_Code := 1;
            L_Selected_Source_Text := 'room';
            L_Selected_Confidence := L_Room_Confidence;
            L_Source_Degraded := TRUE;
            L_Reason_Code := 2;
            L_Reason_Text := 'Room source degraded but retained; floor source unavailable';
        ELSE
            L_Sensor_Error := TRUE;
        END_IF;
    ELSE
        L_Primary_Source_Code := 2; // floor
        L_Primary_Confidence := L_Floor_Confidence;
        L_Fallback_Confidence := L_Room_Confidence;

        // Primary: floor temperature. If floor quality is degraded and room
        // source is healthier, prefer room fallback without declaring hard fault.
        IF L_Floor_Source_Valid AND
           ((L_Floor_Confidence >= L_Min_Source_Confidence) OR NOT L_Room_Source_Valid OR (L_Floor_Confidence >= L_Room_Confidence)) THEN
            L_Current_Temp := fbFloorTempValidator[L_i].VO_Value;
            L_Selected_Source_Code := 2;
            L_Selected_Source_Text := 'floor';
            L_Selected_Confidence := L_Floor_Confidence;
        ELSIF L_Room_Source_Valid THEN
            L_Current_Temp := fbRoomTempValidator[L_Climate_Zone_ID].VO_Value;
            L_Selected_Source_Code := 1;
            L_Selected_Source_Text := 'room';
            L_Selected_Confidence := L_Room_Confidence;
            L_Fallback_Active := TRUE;
        ELSIF L_Floor_Source_Valid THEN
            L_Current_Temp := fbFloorTempValidator[L_i].VO_Value;
            L_Selected_Source_Code := 2;
            L_Selected_Source_Text := 'floor';
            L_Selected_Confidence := L_Floor_Confidence;
            L_Source_Degraded := TRUE;
            L_Reason_Code := 2;
            L_Reason_Text := 'Floor source degraded but retained; room source unavailable';
        ELSE
            L_Sensor_Error := TRUE;
        END_IF;
    END_IF;

    IF L_Fallback_Active THEN
        L_Source_Degraded := TRUE;
        L_Reason_Code := 1;
        IF L_Primary_Source_Code = 1 THEN
            L_Reason_Text := 'Room source degraded or unavailable; floor fallback selected';
        ELSE
            L_Reason_Text := 'Floor source degraded or unavailable; room fallback selected';
        END_IF;
    END_IF;

    IF L_Sensor_Error THEN
        L_Source_Degraded := TRUE;
        L_Reason_Code := 3;
        L_Reason_Text := 'No valid temperature source available';
        VO_Heating_Sensor_Fault := TRUE;
        VO_Zone_Valves[L_i] := FALSE;
    ELSE
        L_Zone_Config := VI_Zone_Configs[L_i];

        IF L_Zone_Config.comfort_temp > REAL#0.0 THEN
            L_Comfort_Target := L_Zone_Config.comfort_temp;
        ELSE
            L_Comfort_Target := L_Zone_Config.design_temp;
        END_IF;

        IF L_Zone_Config.economy_temp > REAL#0.0 THEN
            L_Economy_Target := L_Zone_Config.economy_temp;
        ELSE
            L_Economy_Target := L_Comfort_Target - REAL#3.0;
        END_IF;

        IF L_Zone_Config.long_away_temp > REAL#0.0 THEN
            L_Long_Away_Target := L_Zone_Config.long_away_temp;
        ELSE
            L_Long_Away_Target := GVL_POLICY.G_Away_Long_Economy_Setpoint_C;
        END_IF;

        L_Effective_Target := L_Comfort_Target;

        // Unused rooms may stay in economy even in normal mode.
        IF NOT L_Zone_Config.use_in_normal THEN
            L_Effective_Target := L_Economy_Target;
        END_IF;

        IF GVL_POLICY.G_Away_Active THEN
            CASE GVL_POLICY.G_Away_Level OF
                1:
                    IF L_Zone_Config.use_in_normal THEN
                        L_Effective_Target := L_Comfort_Target + GVL_POLICY.G_Away_Heating_Offset_C;
                    ELSE
                        L_Effective_Target := L_Economy_Target;
                    END_IF;
                2:
                    L_Effective_Target := L_Economy_Target;
                3:
                    L_Effective_Target := L_Long_Away_Target;
            ELSE
                    ;
            END_CASE;

            // Planned return preheat warms only rooms selected in configuration.
            IF GVL_POLICY.G_Away_Return_Preheat_Active AND L_Zone_Config.use_in_away_preheat THEN
                L_Effective_Target := L_Comfort_Target;
            END_IF;
        END_IF;

        IF (L_Climate_Zone_ID >= 1) AND (L_Climate_Zone_ID <= GVL_CONSTANTS.C_MAX_ZONES) THEN
            L_Effective_Target := L_Effective_Target + GVL_HEATING_POLICY.G_Zone_Target_Adjustment[L_Climate_Zone_ID];
        END_IF;

        L_Effective_Target := L_Effective_Target + VI_Scenario_Adjust;

        L_Max_Target := L_Zone_Config.max_temp;
        IF L_Max_Target <= REAL#0.0 THEN
            L_Max_Target := REAL#45.0;
        END_IF;

        IF L_Effective_Target < REAL#5.0 THEN
            L_Effective_Target := REAL#5.0;
        ELSIF L_Effective_Target > L_Max_Target THEN
            L_Effective_Target := L_Max_Target;
        END_IF;

        L_Zone_Config.design_temp := L_Effective_Target;

        L_Floor_Controllers[L_i](
            VI_Current_Temp := L_Current_Temp,
            VI_Config := L_Zone_Config,
            VI_Tariff := VI_Tariff,
            VI_Current_Hour := VI_Current_Hour,
            VI_IsActivePLC := VI_IsActivePLC,
            VI_System_Time_MS := VI_System_Time_MS,
            VO_Valve_Bool => VO_Zone_Valves[L_i]
        );
    END_IF;

    L_Source_Loss_Active := L_Sensor_Error;

    L_Source_Switched_Event :=
        (L_Prev_Selected_Source_Code[L_i] <> 0) AND
        (L_Selected_Source_Code <> 0) AND
        (L_Selected_Source_Code <> L_Prev_Selected_Source_Code[L_i]);

    L_Fallback_Activated_Event :=
        L_Fallback_Active AND NOT L_Prev_Fallback_Active[L_i];

    L_Fallback_Recovered_Event :=
        (NOT L_Fallback_Active) AND L_Prev_Fallback_Active[L_i] AND NOT L_Source_Loss_Active;

    L_Source_Loss_Event :=
        L_Source_Loss_Active AND NOT L_Prev_Source_Loss[L_i];

    L_Last_Event_Code := 0;
    L_Last_Event_Text := '';

    IF L_Source_Loss_Event THEN
        L_Last_Event_Code := 4;
        L_Last_Event_Text := 'Temperature source loss';
    ELSIF L_Fallback_Activated_Event THEN
        L_Last_Event_Code := 2;
        L_Last_Event_Text := L_Reason_Text;
    ELSIF L_Fallback_Recovered_Event THEN
        L_Last_Event_Code := 3;
        L_Last_Event_Text := 'Fallback recovered; primary source selected';
    ELSIF L_Source_Switched_Event THEN
        L_Last_Event_Code := 1;
        L_Last_Event_Text := 'Temperature source switched';
    END_IF;

    GVL_Heating_Runtime_Projection.G_Circuit_Projection[L_i].Visible := TRUE;
    GVL_Heating_Runtime_Projection.G_Circuit_Projection[L_i].Selected_Source_Code := L_Selected_Source_Code;
    GVL_Heating_Runtime_Projection.G_Circuit_Projection[L_i].Selected_Source_Confidence := L_Selected_Confidence;
    GVL_Heating_Runtime_Projection.G_Circuit_Projection[L_i].Fallback_Active := L_Fallback_Active;
    GVL_Heating_Runtime_Projection.G_Circuit_Projection[L_i].Source_Degraded := L_Source_Degraded;
    GVL_Heating_Runtime_Projection.G_Circuit_Projection[L_i].Sensor_Error_Active := L_Sensor_Error;
    GVL_Heating_Runtime_Projection.G_Circuit_Projection[L_i].Reason_Code := L_Reason_Code;
    GVL_Heating_Runtime_Projection.G_Circuit_Projection[L_i].Reason_Text := L_Reason_Text;
    GVL_Heating_Runtime_Projection.G_Circuit_Projection[L_i].Source_Switched_Event := L_Source_Switched_Event;
    GVL_Heating_Runtime_Projection.G_Circuit_Projection[L_i].Fallback_Activated_Event := L_Fallback_Activated_Event;
    GVL_Heating_Runtime_Projection.G_Circuit_Projection[L_i].Fallback_Recovered_Event := L_Fallback_Recovered_Event;
    GVL_Heating_Runtime_Projection.G_Circuit_Projection[L_i].Source_Loss_Event := L_Source_Loss_Event;
    GVL_Heating_Runtime_Projection.G_Circuit_Projection[L_i].Last_Event_Code := L_Last_Event_Code;
    GVL_Heating_Runtime_Projection.G_Circuit_Projection[L_i].Last_Event_Text := L_Last_Event_Text;

    IF L_Last_Event_Code <> 0 THEN
        GVL_Heating_Runtime_Projection.G_Circuit_Projection[L_i].Last_Event_MS := VI_System_Time_MS;
    END_IF;

    L_Prev_Selected_Source_Code[L_i] := L_Selected_Source_Code;
    L_Prev_Fallback_Active[L_i] := L_Fallback_Active;
    L_Prev_Source_Loss[L_i] := L_Source_Loss_Active;

    IF L_Overheat_Timer[L_i].Q THEN
        VO_Zone_Valves[L_i] := FALSE;
    END_IF;

    FOR L_j := 1 TO GVL_CONSTANTS.C_MAX_RULES DO
        IF VI_Rule_Actions[L_j].Active AND VI_Rule_Actions[L_j].Target_ID = L_i THEN
            IF VI_Rule_Actions[L_j].Action_Type = E_Rule_Action_Type.ACTION_SET_FLOOR_HEATING THEN
                VO_Zone_Valves[L_i] := (VI_Rule_Actions[L_j].Value > REAL#0.5);
            END_IF;
        END_IF;
    END_FOR;
END_FOR;

// >>> BULK_SYNC_ANCHOR: FB_Heating_Circuit_Control <<<
END_FUNCTION_BLOCK

(* ---- FB_Heating_Manifold_Control.st ---- *)
// ==============================================================================
// Heating manifold control helper
// Internal refactoring helper for FB_Heating_System_Manager.
// Valve test override remains in FB_Heating_System_Manager for now.
// ==============================================================================
FUNCTION_BLOCK FB_Heating_Manifold_Control
VAR_INPUT
    VI_System_Time_MS : UDINT;
    VI_IsActivePLC : BOOL;
    VI_DHW_Heating_Demand : BOOL;
    VI_Freeze_Mode_Active : BOOL;
    VI_Target_Supply_Temp : REAL;
    VI_Any_Zone_Active : ARRAY[1..GVL_CONSTANTS.C_MAX_MANIFOLDS] OF BOOL;
END_VAR

VAR_IN_OUT
    VI_Manifold_Pressures : ARRAY[1..GVL_CONSTANTS.C_MAX_MANIFOLDS] OF REAL;
    VI_Manifold_Currents : ARRAY[1..GVL_CONSTANTS.C_MAX_MANIFOLDS] OF REAL;
    VI_Manifold_Temps_Supply : ARRAY[1..GVL_CONSTANTS.C_MAX_MANIFOLDS] OF REAL;
    VI_Manifold_Temps_Return : ARRAY[1..GVL_CONSTANTS.C_MAX_MANIFOLDS] OF REAL;
END_VAR

VAR_OUTPUT
    VO_Manifold_Pumps : ARRAY[1..GVL_CONSTANTS.C_MAX_MANIFOLDS] OF BOOL;
    VO_Manifold_Valves : ARRAY[1..GVL_CONSTANTS.C_MAX_MANIFOLDS] OF REAL;
    VO_Status : ARRAY[1..GVL_CONSTANTS.C_MAX_MANIFOLDS] OF ST_Manifold_Status;
END_VAR

VAR
    L_i : INT;
    L_Delta_T : REAL;
    L_Status : ST_Manifold_Status;
    L_Empty_Status : ST_Manifold_Status;
    L_PID_Valves : ARRAY[1..GVL_CONSTANTS.C_MAX_MANIFOLDS] OF FB_PID_Controller;
    L_PID_Timer : ARRAY[1..GVL_CONSTANTS.C_MAX_MANIFOLDS] OF FB_System_Timer;
    L_Pump_Run_Timer : ARRAY[1..GVL_CONSTANTS.C_MAX_MANIFOLDS] OF FB_System_Timer;
    L_Pump_Pause_Timer : ARRAY[1..GVL_CONSTANTS.C_MAX_MANIFOLDS] OF FB_System_Timer;
    L_Pump_In_Pause : ARRAY[1..GVL_CONSTANTS.C_MAX_MANIFOLDS] OF BOOL;
    L_Pump_Diag : ARRAY[1..GVL_CONSTANTS.C_MAX_MANIFOLDS] OF FB_Device_Predictive_Diag;
END_VAR

FOR L_i := 1 TO GVL_CONSTANTS.C_MAX_MANIFOLDS DO
    L_Status := L_Empty_Status;

    L_PID_Timer[L_i](IN := TRUE, PT := T#1s, VI_System_Time_MS := VI_System_Time_MS);
    IF L_PID_Timer[L_i].Q THEN
        L_PID_Timer[L_i](IN := FALSE, PT := T#1s, VI_System_Time_MS := VI_System_Time_MS);
        L_PID_Timer[L_i](IN := TRUE, PT := T#1s, VI_System_Time_MS := VI_System_Time_MS);

        L_PID_Valves[L_i](
            VI_SetPoint := VI_Target_Supply_Temp,
            VI_ProcessValue := VI_Manifold_Temps_Supply[L_i],
            VI_Kp := 2.0,
            VI_Tn := 120.0,
            VI_Tv := 0.0,
            VI_Y_Min := 0.0,
            VI_Y_Max := 100.0,
            VI_Cycle_Time_S := 1.0,
            VO_Output => VO_Manifold_Valves[L_i]
        );
    END_IF;

    L_Pump_Run_Timer[L_i](
        IN := VO_Manifold_Pumps[L_i] AND NOT L_Pump_In_Pause[L_i],
        PT := T#72h,
        VI_System_Time_MS := VI_System_Time_MS
    );
    IF L_Pump_Run_Timer[L_i].Q THEN
        L_Pump_In_Pause[L_i] := TRUE;
    END_IF;

    L_Pump_Pause_Timer[L_i](
        IN := L_Pump_In_Pause[L_i],
        PT := T#1h,
        VI_System_Time_MS := VI_System_Time_MS
    );
    IF L_Pump_Pause_Timer[L_i].Q THEN
        L_Pump_In_Pause[L_i] := FALSE;
    END_IF;

    IF VI_DHW_Heating_Demand THEN
        VO_Manifold_Pumps[L_i] := FALSE;
        VO_Manifold_Valves[L_i] := 0.0;
    ELSE
        VO_Manifold_Pumps[L_i] := VI_IsActivePLC AND VI_Any_Zone_Active[L_i] AND NOT L_Pump_In_Pause[L_i];
        IF NOT VO_Manifold_Pumps[L_i] AND NOT VI_Freeze_Mode_Active THEN
            VO_Manifold_Valves[L_i] := 0.0;
        END_IF;
    END_IF;

    IF VI_Freeze_Mode_Active THEN
        VO_Manifold_Pumps[L_i] := TRUE;
        IF VO_Manifold_Valves[L_i] < 35.0 THEN
            VO_Manifold_Valves[L_i] := 35.0;
        END_IF;
    END_IF;

    L_Status.Pump_On := VO_Manifold_Pumps[L_i];
    L_Status.Pump_Current := VI_Manifold_Currents[L_i];
    L_Status.Pressure := VI_Manifold_Pressures[L_i];
    L_Status.Temp_Supply := VI_Manifold_Temps_Supply[L_i];
    L_Status.Temp_Return := VI_Manifold_Temps_Return[L_i];
    L_Status.Valve_Pos := VO_Manifold_Valves[L_i];

    L_Pump_Diag[L_i](
        VI_Current_Value := VI_Manifold_Currents[L_i],
        VI_Nominal_Value := 0.55,
        VI_Is_Running := VO_Manifold_Pumps[L_i],
        VI_Reset_Stats := FALSE,
        VI_System_Time_MS := VI_System_Time_MS,
        VIO_Health_Data := L_Status.Health
    );

    IF VO_Manifold_Pumps[L_i] THEN
        L_Delta_T := VI_Manifold_Temps_Supply[L_i] - VI_Manifold_Temps_Return[L_i];

        L_Status.Error := FALSE;
        L_Status.Error_ID := 0;

        IF VI_Manifold_Currents[L_i] <= 0.01 THEN
            L_Status.Error := TRUE;
            L_Status.Error_ID := TO_WORD(GVL_CONFIG.ERR_PUMP_NO_CURRENT);
        ELSIF VI_Manifold_Currents[L_i] < 0.3 THEN
            L_Status.Error := TRUE;
            L_Status.Error_ID := TO_WORD(GVL_CONFIG.ERR_PUMP_UNDERCURRENT);
        ELSIF VI_Manifold_Currents[L_i] > 1.5 THEN
            L_Status.Error := TRUE;
            L_Status.Error_ID := TO_WORD(GVL_CONFIG.ERR_PUMP_OVERCURRENT);
        END_IF;

        IF (NOT L_Status.Error) AND ((VI_Manifold_Pressures[L_i] < 1.5) OR (VI_Manifold_Pressures[L_i] > 2.5)) THEN
            L_Status.Error := TRUE;
            L_Status.Error_ID := TO_WORD(GVL_CONFIG.ERR_PRESSURE_OUT_OF_RANGE);
        END_IF;

        IF NOT L_Status.Error THEN
            IF L_Delta_T < 5.0 THEN
                L_Status.Error := TRUE;
                L_Status.Error_ID := TO_WORD(GVL_CONFIG.ERR_DELTA_T_LOW);
            ELSIF L_Delta_T > 10.0 THEN
                L_Status.Error := TRUE;
                L_Status.Error_ID := TO_WORD(GVL_CONFIG.ERR_DELTA_T_HIGH);
            END_IF;
        END_IF;
    END_IF;

    VO_Status[L_i] := L_Status;
END_FOR;

// >>> BULK_SYNC_ANCHOR: FB_Heating_Manifold_Control <<<
END_FUNCTION_BLOCK

(* ---- FB_Heating_Optimizer.st ---- *)
FUNCTION_BLOCK FB_Heating_Optimizer
VAR
    L_i : INT;
    L_Load : REAL;
    L_Total_Demand : REAL;
END_VAR

// ==============================================================================
// Ownership note
// ------------------------------------------------------------------------------
// This block calculates optimization diagnostics only.
// It does NOT modify thermal demand.
//
// Thermal demand ownership remains in:
// FB_Heating_Thermal_Model.
// ==============================================================================

L_Total_Demand := 0.0;

// Aggregate thermal load estimate.
FOR L_i := 1 TO GVL_CONSTANTS.C_MAX_ZONES DO
    L_Total_Demand := L_Total_Demand + ABS(GVL_HEATING_POLICY.G_Zone_Thermal_Demand[L_i]);
END_FOR;

GVL_HEATING_POLICY.G_Optimization_Load_Index := L_Total_Demand;
GVL_HEATING_POLICY.G_Optimization_Energy_Saving_Active := FALSE;

// Zone optimization diagnostics.
FOR L_i := 1 TO GVL_CONSTANTS.C_MAX_ZONES DO

    IF L_Total_Demand > 0.01 THEN
        L_Load := ABS(GVL_HEATING_POLICY.G_Zone_Thermal_Demand[L_i]) / L_Total_Demand;
    ELSE
        L_Load := 0.0;
    END_IF;

    GVL_HEATING_POLICY.G_Zone_Optimization_Score[L_i] :=
        L_Load +
        ((1.0 - GVL_HEATING_POLICY.G_Zone_Thermal_Model_Confidence[L_i]) * 0.2);

    // Advisory energy-saving indication only.
    IF L_Total_Demand > 5.0 THEN
        GVL_HEATING_POLICY.G_Optimization_Energy_Saving_Active := TRUE;
    END_IF;

END_FOR;

END_FUNCTION_BLOCK

(* ---- FB_Heating_Policy_Manager.st ---- *)
FUNCTION_BLOCK FB_Heating_Policy_Manager
VAR_INPUT
    VI_System_Time_MS : UDINT;
    VI_System_Mode : E_System_Operating_Mode;
    VI_RootCause : E_Heating_RootCause;
    VI_RootConfidence : REAL;
    VI_Min_Hold_MS : UDINT;
    VI_Emergency_Stop : BOOL;
    VI_Gas_Safety : BOOL;
    VI_Room_Temp_Avg : REAL;
    VI_Floor_Temp_Avg : REAL;
    VI_Supply_Temp : REAL;
    VI_Return_Temp : REAL;
    VI_Target_Temp : REAL;
    VI_Room_Temps : ARRAY[1..GVL_CONSTANTS.C_MAX_ZONES] OF REAL;
    VI_Floor_Temps : ARRAY[1..GVL_CONSTANTS.C_MAX_ZONES] OF REAL;
END_VAR
VAR_OUTPUT
    VO_Policy_Mode : E_Heating_Policy_Mode;
    VO_Block_Heating : BOOL;
    VO_Target_Adjustment : REAL;
    VO_Priority_Multiplier : REAL;
    VO_Self_Tune_Active : BOOL;
    VO_Self_Tune_Level : INT;
    VO_Feedback_Stable : BOOL;
    VO_Feedback_Improving : BOOL;
    VO_Feedback_Quality : REAL;
END_VAR
VAR
    L_Raw_Mode : E_Heating_Policy_Mode;
    L_Raw_Block : BOOL;
    L_Raw_Target_Adjustment : REAL;
    L_Raw_Priority_Multiplier : REAL;
    L_Held_Mode : E_Heating_Policy_Mode;
    L_Held_Block : BOOL;
    L_Held_Target_Adjustment : REAL;
    L_Held_Priority_Multiplier : REAL;
    L_Last_Accept_MS : UDINT;
    L_Initialized : BOOL;
    L_Quality_Initialized : BOOL;
    L_Effective_Hold_MS : UDINT;
    L_Force_Immediate : BOOL;
    L_Same_Cause_Since : UDINT;
    L_Last_Cause : E_Heating_RootCause;
    L_Self_Level : INT;
    L_Room_Error : REAL;
    L_Supply_Error : REAL;
    L_DeltaT : REAL;
    L_Quality : REAL;
    L_Last_Quality : REAL;
    L_Improving : BOOL;
    L_Stable : BOOL;
    L_Last_Room_Avg : REAL;
    L_Trend : REAL;
    L_Filtered_Trend : REAL;
    L_Predictive_Adjustment : REAL;
    L_i : INT;
    L_Zone_Error : REAL;
    L_Zone_Quality : REAL;
    L_Zone_Desired_Level : INT;
    L_Zone_Last_Level_Accept_MS : ARRAY[1..GVL_CONSTANTS.C_MAX_ZONES] OF UDINT;
    L_Zone_Hold_MS : UDINT;
END_VAR

// ==============================================================================
// Ownership note
// ------------------------------------------------------------------------------
// This block owns only global policy mode/adjustment and policy quality/self-tune
// diagnostics. It does NOT own per-zone thermal fields, per-zone target adjustment,
// preheat request, or optimization demand values.
//
// Field owners:
// - FB_Heating_Thermal_Model: thermal response/demand/time/model confidence;
// - FB_Heating_Predictive_Controller: preheat-needed prediction;
// - FB_Heating_Optimizer: optimization scores/load diagnostics;
// - FB_Heating_Policy_Observer / FB_Heating_Schedule_Preheat: zone target policy;
// - FB_Heating_Policy_Manager: global policy and quality/self-level diagnostics.
// ==============================================================================

L_Zone_Hold_MS := VI_Min_Hold_MS / 2;
IF L_Zone_Hold_MS < 60000 THEN
    L_Zone_Hold_MS := 60000;
END_IF;

IF NOT L_Quality_Initialized THEN
    L_Last_Room_Avg := VI_Room_Temp_Avg;
    L_Filtered_Trend := 0.0;
    L_Same_Cause_Since := VI_System_Time_MS;
    L_Last_Cause := VI_RootCause;

    FOR L_i := 1 TO GVL_CONSTANTS.C_MAX_ZONES DO
        L_Zone_Last_Level_Accept_MS[L_i] := VI_System_Time_MS;
        GVL_HEATING_POLICY.G_Zone_Quality[L_i] := 0.0;
        GVL_HEATING_POLICY.G_Zone_Improving[L_i] := FALSE;
        GVL_HEATING_POLICY.G_Zone_Stable[L_i] := TRUE;
        GVL_HEATING_POLICY.G_Zone_Self_Level[L_i] := 0;
    END_FOR;

    L_Quality_Initialized := TRUE;
END_IF;

// ==============================================================================
// Global predictive adjustment based on aggregate room trend.
// ==============================================================================
L_Trend := VI_Room_Temp_Avg - L_Last_Room_Avg;
L_Last_Room_Avg := VI_Room_Temp_Avg;
L_Filtered_Trend := (L_Filtered_Trend * 0.8) + (L_Trend * 0.2);

L_Predictive_Adjustment := 0.0;
IF (L_Filtered_Trend < -0.03) AND (VI_Room_Temp_Avg < (VI_Target_Temp + 0.5)) THEN
    L_Predictive_Adjustment := 1.0;
ELSIF L_Filtered_Trend > 0.03 THEN
    L_Predictive_Adjustment := -0.5;
END_IF;

IF L_Predictive_Adjustment > 1.0 THEN
    L_Predictive_Adjustment := 1.0;
END_IF;
IF L_Predictive_Adjustment < -1.0 THEN
    L_Predictive_Adjustment := -1.0;
END_IF;

GVL_HEATING_POLICY.G_Policy_Predictive_Adjustment := L_Predictive_Adjustment;
GVL_HEATING_POLICY.G_Policy_Predictive_Active := ABS(L_Predictive_Adjustment) > 0.001;

// ==============================================================================
// Aggregate quality / feedback diagnostics.
// ==============================================================================
L_Room_Error := VI_Target_Temp - VI_Room_Temp_Avg;
L_Supply_Error := VI_Target_Temp - VI_Supply_Temp;
L_DeltaT := VI_Supply_Temp - VI_Return_Temp;
L_Quality := 0.0;

IF L_Room_Error > 1.0 THEN
    L_Quality := L_Quality + 2.0;
END_IF;
IF L_Supply_Error > 1.0 THEN
    L_Quality := L_Quality + 1.0;
END_IF;
IF L_DeltaT < 3.0 THEN
    L_Quality := L_Quality + 1.0;
END_IF;

L_Improving := L_Quality < L_Last_Quality;
L_Stable := L_Quality = 0.0;

// ==============================================================================
// Per-zone quality / self-level diagnostics only.
// Does not write target adjustment, thermal demand, time-to-heat, or preheat flags.
// ==============================================================================
FOR L_i := 1 TO GVL_CONSTANTS.C_MAX_ZONES DO
    L_Zone_Error := VI_Target_Temp - VI_Room_Temps[L_i];
    L_Zone_Quality := 0.0;

    IF L_Zone_Error > 1.0 THEN
        L_Zone_Quality := L_Zone_Quality + 2.0;
    END_IF;
    IF VI_Floor_Temps[L_i] < (VI_Target_Temp - 2.0) THEN
        L_Zone_Quality := L_Zone_Quality + 1.0;
    END_IF;

    GVL_HEATING_POLICY.G_Zone_Improving[L_i] :=
        L_Zone_Quality < GVL_HEATING_POLICY.G_Zone_Quality[L_i];

    GVL_HEATING_POLICY.G_Zone_Stable[L_i] :=
        L_Zone_Quality = 0.0;

    L_Zone_Desired_Level := GVL_HEATING_POLICY.G_Zone_Self_Level[L_i];

    IF GVL_HEATING_POLICY.G_Zone_Stable[L_i] THEN
        L_Zone_Desired_Level := 0;
    ELSIF GVL_HEATING_POLICY.G_Zone_Improving[L_i] THEN
        L_Zone_Desired_Level := GVL_HEATING_POLICY.G_Zone_Self_Level[L_i] - 1;
    ELSIF L_Zone_Quality >= 3.0 THEN
        L_Zone_Desired_Level := GVL_HEATING_POLICY.G_Zone_Self_Level[L_i] + 1;
    END_IF;

    IF L_Zone_Desired_Level > 2 THEN
        L_Zone_Desired_Level := 2;
    END_IF;
    IF L_Zone_Desired_Level < 0 THEN
        L_Zone_Desired_Level := 0;
    END_IF;

    IF L_Zone_Desired_Level <> GVL_HEATING_POLICY.G_Zone_Self_Level[L_i] THEN
        IF (VI_System_Time_MS - L_Zone_Last_Level_Accept_MS[L_i]) >= L_Zone_Hold_MS THEN
            GVL_HEATING_POLICY.G_Zone_Self_Level[L_i] := L_Zone_Desired_Level;
            L_Zone_Last_Level_Accept_MS[L_i] := VI_System_Time_MS;
        END_IF;
    END_IF;

    GVL_HEATING_POLICY.G_Zone_Quality[L_i] := L_Zone_Quality;
END_FOR;

// ==============================================================================
// Global self-level and policy mode.
// ==============================================================================
IF VI_RootCause <> L_Last_Cause THEN
    L_Same_Cause_Since := VI_System_Time_MS;
    L_Self_Level := 0;
END_IF;
L_Last_Cause := VI_RootCause;

IF L_Stable THEN
    L_Self_Level := 0;
ELSIF L_Improving THEN
    L_Self_Level := L_Self_Level - 1;
ELSIF (VI_System_Time_MS - L_Same_Cause_Since) > (VI_Min_Hold_MS * 2) AND (VI_RootConfidence > 0.8) AND (L_Quality >= 3.0) THEN
    L_Self_Level := L_Self_Level + 1;
END_IF;

IF L_Self_Level > 2 THEN
    L_Self_Level := 2;
END_IF;
IF L_Self_Level < 0 THEN
    L_Self_Level := 0;
END_IF;

L_Raw_Mode := E_Heating_Policy_Mode.HPM_NORMAL;
L_Raw_Block := FALSE;
L_Raw_Target_Adjustment := L_Predictive_Adjustment;
L_Raw_Priority_Multiplier := 1.0;
L_Force_Immediate := FALSE;

IF VI_Emergency_Stop OR VI_Gas_Safety THEN
    L_Raw_Mode := E_Heating_Policy_Mode.HPM_SAFETY_BLOCK;
    L_Raw_Block := TRUE;
    L_Raw_Target_Adjustment := 0.0;
    L_Raw_Priority_Multiplier := 1.0;
    L_Force_Immediate := TRUE;
ELSIF VI_RootCause = E_Heating_RootCause.RC_IO_OFFLINE THEN
    L_Raw_Mode := E_Heating_Policy_Mode.HPM_DEGRADED;
    L_Raw_Block := TRUE;
    L_Raw_Target_Adjustment := 0.0;
    L_Raw_Priority_Multiplier := 1.0;
    L_Force_Immediate := TRUE;
ELSIF VI_RootConfidence >= 0.6 THEN
    CASE VI_RootCause OF
        E_Heating_RootCause.RC_NO_HEAT_TRANSFER:
            L_Raw_Mode := E_Heating_Policy_Mode.HPM_DEGRADED;
            L_Raw_Target_Adjustment := L_Raw_Target_Adjustment + 3.0 + TO_REAL(L_Self_Level);
        E_Heating_RootCause.RC_PUMP_FAILURE:
            L_Raw_Mode := E_Heating_Policy_Mode.HPM_FAULT_ISOLATION;
            L_Raw_Priority_Multiplier := 0.5 - (0.1 * TO_REAL(L_Self_Level));
        E_Heating_RootCause.RC_VALVES_CLOSED:
            L_Raw_Mode := E_Heating_Policy_Mode.HPM_FAULT_ISOLATION;
            L_Raw_Target_Adjustment := L_Raw_Target_Adjustment - 2.0;
        E_Heating_RootCause.RC_NO_FLAME,
        E_Heating_RootCause.RC_BOILER_ERROR:
            L_Raw_Mode := E_Heating_Policy_Mode.HPM_DEGRADED;
            L_Raw_Priority_Multiplier := 0.7;
    ELSE
        IF VI_System_Mode = E_System_Operating_Mode.MODE_DEGRADED THEN
            L_Raw_Mode := E_Heating_Policy_Mode.HPM_DEGRADED;
        END_IF;
    END_CASE;
ELSE
    IF VI_System_Mode = E_System_Operating_Mode.MODE_DEGRADED THEN
        L_Raw_Mode := E_Heating_Policy_Mode.HPM_DEGRADED;
    END_IF;
END_IF;

IF L_Raw_Target_Adjustment > 5.0 THEN
    L_Raw_Target_Adjustment := 5.0;
END_IF;
IF L_Raw_Target_Adjustment < -3.0 THEN
    L_Raw_Target_Adjustment := -3.0;
END_IF;
IF L_Raw_Priority_Multiplier < 0.3 THEN
    L_Raw_Priority_Multiplier := 0.3;
END_IF;
IF L_Raw_Priority_Multiplier > 1.0 THEN
    L_Raw_Priority_Multiplier := 1.0;
END_IF;

L_Effective_Hold_MS := VI_Min_Hold_MS;
IF VI_RootConfidence >= 0.9 THEN
    L_Effective_Hold_MS := VI_Min_Hold_MS / 2;
END_IF;

IF NOT L_Initialized THEN
    L_Held_Mode := L_Raw_Mode;
    L_Held_Block := L_Raw_Block;
    L_Held_Target_Adjustment := L_Raw_Target_Adjustment;
    L_Held_Priority_Multiplier := L_Raw_Priority_Multiplier;
    L_Last_Accept_MS := VI_System_Time_MS;
    L_Initialized := TRUE;
ELSIF L_Force_Immediate THEN
    L_Held_Mode := L_Raw_Mode;
    L_Held_Block := L_Raw_Block;
    L_Held_Target_Adjustment := L_Raw_Target_Adjustment;
    L_Held_Priority_Multiplier := L_Raw_Priority_Multiplier;
    L_Last_Accept_MS := VI_System_Time_MS;
ELSIF (L_Raw_Mode <> L_Held_Mode) OR (ABS(L_Raw_Target_Adjustment - L_Held_Target_Adjustment) > 0.001) OR (ABS(L_Raw_Priority_Multiplier - L_Held_Priority_Multiplier) > 0.001) OR (L_Raw_Block <> L_Held_Block) THEN
    IF (VI_System_Time_MS - L_Last_Accept_MS) >= L_Effective_Hold_MS THEN
        L_Held_Mode := L_Raw_Mode;
        L_Held_Block := L_Raw_Block;
        L_Held_Target_Adjustment := L_Raw_Target_Adjustment;
        L_Held_Priority_Multiplier := L_Raw_Priority_Multiplier;
        L_Last_Accept_MS := VI_System_Time_MS;
    END_IF;
END_IF;

VO_Policy_Mode := L_Held_Mode;
VO_Block_Heating := L_Held_Block;
VO_Target_Adjustment := L_Held_Target_Adjustment;
VO_Priority_Multiplier := L_Held_Priority_Multiplier;
VO_Self_Tune_Active := L_Self_Level > 0;
VO_Self_Tune_Level := L_Self_Level;
VO_Feedback_Stable := L_Stable;
VO_Feedback_Improving := L_Improving;
VO_Feedback_Quality := L_Quality;

L_Last_Quality := L_Quality;

END_FUNCTION_BLOCK

(* ---- FB_Heating_Policy_Observer.st ---- *)
FUNCTION_BLOCK FB_Heating_Policy_Observer

VAR_INPUT
    VI_Zone_Occupied : ARRAY[1..GVL_CONSTANTS.C_MAX_ZONES] OF BOOL;
    VI_Zone_Last_Motion_TS : ARRAY[1..GVL_CONSTANTS.C_MAX_ZONES] OF UDINT;
    VI_System_Time_MS : UDINT;
    VI_Zone_Permanent_Use : ARRAY[1..GVL_CONSTANTS.C_MAX_ZONES] OF BOOL;
    VI_Zone_Guest_Preheat : ARRAY[1..GVL_CONSTANTS.C_MAX_ZONES] OF BOOL;
    VI_Behavior_Mode : E_Behavior_Mode;
END_VAR

VAR_OUTPUT
    VO_Zone_Empty_Duration_MS : ARRAY[1..GVL_CONSTANTS.C_MAX_ZONES] OF UDINT;
    VO_Zone_Policy_Class : ARRAY[1..GVL_CONSTANTS.C_MAX_ZONES] OF INT;
    VO_Zone_Target_Adjustment : ARRAY[1..GVL_CONSTANTS.C_MAX_ZONES] OF REAL;
    VO_Zone_Priority_Bias : ARRAY[1..GVL_CONSTANTS.C_MAX_ZONES] OF REAL;
END_VAR

VAR
    L_i : INT;
    L_Long_Threshold : UDINT := 86400000; // 24h
    L_Away_Mode : BOOL;
END_VAR

L_Away_Mode := (VI_Behavior_Mode = BEHAVIOR_AWAY);

FOR L_i := 1 TO GVL_CONSTANTS.C_MAX_ZONES DO

    // compute empty duration
    IF VI_Zone_Occupied[L_i] THEN
        VO_Zone_Empty_Duration_MS[L_i] := 0;
    ELSE
        VO_Zone_Empty_Duration_MS[L_i] := VI_System_Time_MS - VI_Zone_Last_Motion_TS[L_i];
    END_IF;

    // policy classification
    // Guest/preheat has priority even in AWAY mode.
    IF VI_Zone_Guest_Preheat[L_i] THEN
        VO_Zone_Policy_Class[L_i] := 3; // guest

    ELSIF VI_Zone_Occupied[L_i] THEN
        VO_Zone_Policy_Class[L_i] := 0; // comfort

    ELSIF VI_Zone_Permanent_Use[L_i] AND (NOT L_Away_Mode) THEN
        VO_Zone_Policy_Class[L_i] := 4; // permanent mild eco

    ELSIF VO_Zone_Empty_Duration_MS[L_i] >= L_Long_Threshold THEN
        VO_Zone_Policy_Class[L_i] := 2; // deep eco

    ELSE
        VO_Zone_Policy_Class[L_i] := 1; // mild eco
    END_IF;

    // observe-only target adjustment (no effect yet)
    CASE VO_Zone_Policy_Class[L_i] OF
        0: // comfort
            VO_Zone_Target_Adjustment[L_i] := 0.0;
            VO_Zone_Priority_Bias[L_i] := 1.0;

        1: // mild eco
            VO_Zone_Target_Adjustment[L_i] := -1.0;
            VO_Zone_Priority_Bias[L_i] := 0.8;

        2: // deep eco
            VO_Zone_Target_Adjustment[L_i] := -3.0;
            VO_Zone_Priority_Bias[L_i] := 0.5;

        3: // guest preheat
            VO_Zone_Target_Adjustment[L_i] := 0.0;
            VO_Zone_Priority_Bias[L_i] := 1.5;

        4: // permanent-use mild eco
            VO_Zone_Target_Adjustment[L_i] := -0.5;
            VO_Zone_Priority_Bias[L_i] := 0.9;

    END_CASE;

END_FOR;
END_FUNCTION_BLOCK
